LIN {X 0,Y 573.939,Z 295.271,A -85,B 0,C 180,E1 -2262.554,E2 -2262.554} C_VEL
LIN {X 0,Y 573.907,Z 198.013,A -85,B 0,C 180,E1 -2263.779,E2 -2263.779} C_VEL
LIN {X 0,Y 573.417,Z 194.435,A -85,B 0,C 180,E1 -2263.851,E2 -2263.851} C_VEL
LIN {X 0,Y 573.583,Z 173.354,A -85,B 0,C 180,E1 -2266.732,E2 -2266.732} C_VEL
LIN {X 0,Y 573.724,Z 153.908,A -85,B 0,C 180,E1 -2269.398,E2 -2269.398} C_VEL
LIN {X 0,Y 573.977,Z 134.142,A -85,B 0,C 180,E1 -2272.118,E2 -2272.118} C_VEL
LIN {X 0,Y 573.891,Z 125.743,A -85,B 0,C 180,E1 -2273.296,E2 -2273.296} C_VEL
LIN {X 0,Y 573.251,Z 122.082,A -85,B 0,C 180,E1 -2273.865,E2 -2273.865} C_VEL
LIN {X 0,Y 573.218,Z 122.082,A -85,B 0,C 180,E1 -2276.488,E2 -2276.488} C_VEL
LIN {X 0,Y 573.233,Z 122.079,A -85,B 0,C 180,E1 -2278.565,E2 -2278.565} C_VEL
LIN {X 0,Y 573.222,Z 122.078,A -85,B 0,C 180,E1 -2280.994,E2 -2280.994} C_VEL
LIN {X 0,Y 573.266,Z 122.077,A -85,B 0,C 180,E1 -2283.524,E2 -2283.524} C_VEL
LIN {X 0,Y 573.195,Z 122.085,A -85,B 0,C 180,E1 -2286.053,E2 -2286.053} C_VEL
LIN {X 0,Y 573.244,Z 122.074,A -85,B 0,C 180,E1 -2288.702,E2 -2288.702} C_VEL
LIN {X 0,Y 573.225,Z 122.086,A -85,B 0,C 180,E1 -2291.592,E2 -2291.592} C_VEL
LIN {X 0,Y 573.223,Z 122.077,A -85,B 0,C 180,E1 -2294.335,E2 -2294.335} C_VEL
LIN {X 0,Y 573.237,Z 122.084,A -85,B 0,C 180,E1 -2297.359,E2 -2297.359} C_VEL
LIN {X 0,Y 573.233,Z 122.076,A -85,B 0,C 180,E1 -2300.392,E2 -2300.392} C_VEL
LIN {X 0,Y 573.25,Z 122.082,A -85,B 0,C 180,E1 -2303.077,E2 -2303.077} C_VEL
LIN {X 0,Y 573.25,Z 122.075,A -85,B 0,C 180,E1 -2305.67,E2 -2305.67} C_VEL
LIN {X 0,Y 573.224,Z 122.077,A -85,B 0,C 180,E1 -2308.183,E2 -2308.183} C_VEL
LIN {X 0,Y 573.231,Z 122.081,A -85,B 0,C 180,E1 -2310.632,E2 -2310.632} C_VEL
LIN {X 0,Y 573.211,Z 122.079,A -85,B 0,C 180,E1 -2313.513,E2 -2313.513} C_VEL
LIN {X 0,Y 573.192,Z 122.082,A -85,B 0,C 180,E1 -2316.133,E2 -2316.133} C_VEL
LIN {X 0,Y 573.224,Z 122.078,A -85,B 0,C 180,E1 -2319.173,E2 -2319.173} C_VEL
LIN {X 0,Y 573.189,Z 122.08,A -85,B 0,C 180,E1 -2321.41,E2 -2321.41} C_VEL
LIN {X 0,Y 573.199,Z 122.088,A -85,B 0,C 180,E1 -2324.351,E2 -2324.351} C_VEL
LIN {X 0,Y 573.188,Z 122.088,A -85,B 0,C 180,E1 -2326.528,E2 -2326.528} C_VEL
LIN {X 0,Y 573.233,Z 122.075,A -85,B 0,C 180,E1 -2329.403,E2 -2329.403} C_VEL
LIN {X 0,Y 573.209,Z 122.087,A -85,B 0,C 180,E1 -2332.249,E2 -2332.249} C_VEL
LIN {X 0,Y 573.266,Z 122.071,A -85,B 0,C 180,E1 -2335.077,E2 -2335.077} C_VEL
LIN {X 0,Y 573.306,Z 122.073,A -85,B 0,C 180,E1 -2337.892,E2 -2337.892} C_VEL
LIN {X 0,Y 573.314,Z 122.073,A -85,B 0,C 180,E1 -2340,E2 -2340} C_VEL
LIN {X 0,Y 573.268,Z 122.069,A -85,B 0,C 180,E1 -2342.811,E2 -2342.811} C_VEL
LIN {X 0,Y 573.27,Z 122.079,A -85,B 0,C 180,E1 -2345.628,E2 -2345.628} C_VEL
LIN {X 0,Y 573.241,Z 122.073,A -85,B 0,C 180,E1 -2348.46,E2 -2348.46} C_VEL
LIN {X 0,Y 573.271,Z 122.077,A -85,B 0,C 180,E1 -2351.312,E2 -2351.312} C_VEL
LIN {X 0,Y 573.253,Z 122.071,A -85,B 0,C 180,E1 -2354.413,E2 -2354.413} C_VEL
LIN {X 0,Y 573.245,Z 122.08,A -85,B 0,C 180,E1 -2357.112,E2 -2357.112} C_VEL
LIN {X 0,Y 573.232,Z 122.075,A -85,B 0,C 180,E1 -2360.078,E2 -2360.078} C_VEL
LIN {X 0,Y 573.22,Z 122.077,A -85,B 0,C 180,E1 -2362.339,E2 -2362.339} C_VEL
LIN {X 0,Y 573.198,Z 122.079,A -85,B 0,C 180,E1 -2364.344,E2 -2364.344} C_VEL
LIN {X 0,Y 572.559,Z 122.166,A -85,B 0,C 180,E1 -2364.931,E2 -2364.931} C_VEL
LIN {X 0,Y 569.731,Z 122.52,A -85,B 0,C 180,E1 -2365.883,E2 -2365.883} C_VEL
LIN {X 0,Y 567.32,Z 122.82,A -85,B 0,C 180,E1 -2366.648,E2 -2366.648} C_VEL
LIN {X 0,Y 566.274,Z 122.948,A -85,B 0,C 180,E1 -2367.239,E2 -2367.239} C_VEL
LIN {X 0,Y 566.184,Z 122.956,A -85,B 0,C 180,E1 -2367.44,E2 -2367.44} C_VEL
LIN {X 0,Y 566.172,Z 122.955,A -85,B 0,C 180,E1 -2369.771,E2 -2369.771} C_VEL
LIN {X 0,Y 566.201,Z 122.955,A -85,B 0,C 180,E1 -2372.43,E2 -2372.43} C_VEL
LIN {X 0,Y 566.18,Z 122.959,A -85,B 0,C 180,E1 -2374.989,E2 -2374.989} C_VEL
LIN {X 0,Y 566.197,Z 122.952,A -85,B 0,C 180,E1 -2377.461,E2 -2377.461} C_VEL
LIN {X 0,Y 566.208,Z 122.954,A -85,B 0,C 180,E1 -2380.199,E2 -2380.199} C_VEL
LIN {X 0,Y 566.2,Z 122.953,A -85,B 0,C 180,E1 -2383.055,E2 -2383.055} C_VEL
LIN {X 0,Y 566.196,Z 122.957,A -85,B 0,C 180,E1 -2386.049,E2 -2386.049} C_VEL
LIN {X 0,Y 566.206,Z 122.951,A -85,B 0,C 180,E1 -2389.215,E2 -2389.215} C_VEL
LIN {X 0,Y 566.189,Z 122.956,A -85,B 0,C 180,E1 -2391.637,E2 -2391.637} C_VEL
LIN {X 0,Y 566.165,Z 122.962,A -85,B 0,C 180,E1 -2394.308,E2 -2394.308} C_VEL
LIN {X 0,Y 566.224,Z 122.949,A -85,B 0,C 180,E1 -2396.898,E2 -2396.898} C_VEL
LIN {X 0,Y 566.184,Z 122.957,A -85,B 0,C 180,E1 -2399.407,E2 -2399.407} C_VEL
LIN {X 0,Y 566.198,Z 122.961,A -85,B 0,C 180,E1 -2401.856,E2 -2401.856} C_VEL
LIN {X 0,Y 566.217,Z 122.953,A -85,B 0,C 180,E1 -2404.251,E2 -2404.251} C_VEL
LIN {X 0,Y 566.24,Z 123.02,A -85,B 0,C 180,E1 -2406.598,E2 -2406.598} C_VEL
LIN {X 0,Y 566.394,Z 130.26,A -85,B 0,C 180,E1 -2407.954,E2 -2407.954} C_VEL
LIN {X 0,Y 566.229,Z 145.729,A -85,B 0,C 180,E1 -2410.874,E2 -2410.874} C_VEL
LIN {X 0,Y 566.186,Z 146.658,A -85,B 0,C 180,E1 -2411.05,E2 -2411.05} C_VEL
LIN {X 0,Y 567.206,Z 153.44,A -85,B 0,C 180,E1 -2411.169,E2 -2411.169} C_VEL
LIN {X 0,Y 566.897,Z 253.478,A -85,B 0,C 180,E1 -2412.457,E2 -2412.457} C_VEL
LIN {X 0,Y 566.788,Z 267.319,A -85,B 0,C 180,E1 -2412.796,E2 -2412.796} C_VEL
LIN {X 0,Y 566.722,Z 279.942,A -85,B 0,C 180,E1 -2413.258,E2 -2413.258} C_VEL
LIN {X 0,Y 566.568,Z 292.491,A -85,B 0,C 180,E1 -2413.885,E2 -2413.885} C_VEL
LIN {X 0,Y 566.436,Z 303.91,A -85,B 0,C 180,E1 -2414.62,E2 -2414.62} C_VEL
LIN {X 0,Y 566.278,Z 314.5,A -85,B 0,C 180,E1 -2415.479,E2 -2415.479} C_VEL
LIN {X 0,Y 566.22,Z 323.325,A -85,B 0,C 180,E1 -2416.359,E2 -2416.359} C_VEL
LIN {X 0,Y 566.067,Z 332.259,A -85,B 0,C 180,E1 -2417.451,E2 -2417.451} C_VEL
LIN {X 0,Y 566.016,Z 339.371,A -85,B 0,C 180,E1 -2418.541,E2 -2418.541} C_VEL
LIN {X 0,Y 565.933,Z 345.026,A -85,B 0,C 180,E1 -2419.626,E2 -2419.626} C_VEL
LIN {X 0,Y 565.88,Z 349.456,A -85,B 0,C 180,E1 -2420.708,E2 -2420.708} C_VEL
LIN {X 0,Y 565.891,Z 351.793,A -85,B 0,C 180,E1 -2421.429,E2 -2421.429} C_VEL
LIN {X 0,Y 565.891,Z 353.691,A -85,B 0,C 180,E1 -2422.148,E2 -2422.148} C_VEL
LIN {X 0,Y 565.923,Z 356.006,A -85,B 0,C 180,E1 -2423.463,E2 -2423.463} C_VEL
LIN {X 0,Y 565.899,Z 356.763,A -85,B 0,C 180,E1 -2424.297,E2 -2424.297} C_VEL
LIN {X 0,Y 565.849,Z 356.998,A -85,B 0,C 180,E1 -2425.012,E2 -2425.012} C_VEL
LIN {X 0,Y 565.912,Z 356.806,A -85,B 0,C 180,E1 -2425.726,E2 -2425.726} C_VEL
LIN {X 0,Y 565.911,Z 356.216,A -85,B 0,C 180,E1 -2426.439,E2 -2426.439} C_VEL
LIN {X 0,Y 565.841,Z 353.871,A -85,B 0,C 180,E1 -2427.864,E2 -2427.864} C_VEL
LIN {X 0,Y 565.888,Z 350.984,A -85,B 0,C 180,E1 -2428.932,E2 -2428.932} C_VEL
LIN {X 0,Y 565.905,Z 347.081,A -85,B 0,C 180,E1 -2429.999,E2 -2429.999} C_VEL
LIN {X 0,Y 565.991,Z 342.057,A -85,B 0,C 180,E1 -2431.067,E2 -2431.067} C_VEL
LIN {X 0,Y 565.977,Z 335.764,A -85,B 0,C 180,E1 -2432.134,E2 -2432.134} C_VEL
LIN {X 0,Y 566.169,Z 327.896,A -85,B 0,C 180,E1 -2433.201,E2 -2433.201} C_VEL
LIN {X 0,Y 566.237,Z 319.912,A -85,B 0,C 180,E1 -2434.092,E2 -2434.092} C_VEL
LIN {X 0,Y 566.321,Z 310.198,A -85,B 0,C 180,E1 -2434.983,E2 -2434.983} C_VEL
LIN {X 0,Y 566.461,Z 299.366,A -85,B 0,C 180,E1 -2435.785,E2 -2435.785} C_VEL
LIN {X 0,Y 566.658,Z 287.581,A -85,B 0,C 180,E1 -2436.47,E2 -2436.47} C_VEL
LIN {X 0,Y 566.766,Z 275.517,A -85,B 0,C 180,E1 -2437.011,E2 -2437.011} C_VEL
LIN {X 0,Y 566.847,Z 263.545,A -85,B 0,C 180,E1 -2437.405,E2 -2437.405} C_VEL
LIN {X 0,Y 566.903,Z 250.677,A -85,B 0,C 180,E1 -2437.68,E2 -2437.68} C_VEL
LIN {X 0,Y 567.048,Z 151.584,A -85,B 0,C 180,E1 -2438.949,E2 -2438.949} C_VEL
LIN {X 0,Y 566.192,Z 146.551,A -85,B 0,C 180,E1 -2439.06,E2 -2439.06} C_VEL
LIN {X 0,Y 566.372,Z 131.992,A -85,B 0,C 180,E1 -2441.814,E2 -2441.814} C_VEL
LIN {X 0,Y 566.232,Z 122.953,A -85,B 0,C 180,E1 -2443.525,E2 -2443.525} C_VEL
LIN {X 0,Y 566.213,Z 122.957,A -85,B 0,C 180,E1 -2446.587,E2 -2446.587} C_VEL
LIN {X 0,Y 566.203,Z 122.952,A -85,B 0,C 180,E1 -2449.58,E2 -2449.58} C_VEL
LIN {X 0,Y 566.194,Z 122.957,A -85,B 0,C 180,E1 -2451.861,E2 -2451.861} C_VEL
LIN {X 0,Y 566.218,Z 122.949,A -85,B 0,C 180,E1 -2455.029,E2 -2455.029} C_VEL
LIN {X 0,Y 566.192,Z 122.954,A -85,B 0,C 180,E1 -2457.339,E2 -2457.339} C_VEL
LIN {X 0,Y 566.198,Z 122.959,A -85,B 0,C 180,E1 -2459.768,E2 -2459.768} C_VEL
LIN {X 0,Y 566.2,Z 122.954,A -85,B 0,C 180,E1 -2462.429,E2 -2462.429} C_VEL
LIN {X 0,Y 566.176,Z 122.955,A -85,B 0,C 180,E1 -2464.988,E2 -2464.988} C_VEL
LIN {X 0,Y 566.192,Z 122.959,A -85,B 0,C 180,E1 -2467.46,E2 -2467.46} C_VEL
LIN {X 0,Y 566.204,Z 122.953,A -85,B 0,C 180,E1 -2470.198,E2 -2470.198} C_VEL
LIN {X 0,Y 566.194,Z 122.956,A -85,B 0,C 180,E1 -2473.053,E2 -2473.053} C_VEL
LIN {X 0,Y 566.187,Z 122.955,A -85,B 0,C 180,E1 -2476.048,E2 -2476.048} C_VEL
LIN {X 0,Y 566.196,Z 122.96,A -85,B 0,C 180,E1 -2479.214,E2 -2479.214} C_VEL
LIN {X 0,Y 566.173,Z 122.959,A -85,B 0,C 180,E1 -2481.635,E2 -2481.635} C_VEL
LIN {X 0,Y 566.153,Z 122.958,A -85,B 0,C 180,E1 -2484.307,E2 -2484.307} C_VEL
LIN {X 0,Y 566.189,Z 122.961,A -85,B 0,C 180,E1 -2486.896,E2 -2486.896} C_VEL
LIN {X 0,Y 566.161,Z 122.96,A -85,B 0,C 180,E1 -2489.406,E2 -2489.406} C_VEL
LIN {X 0,Y 566.183,Z 122.954,A -85,B 0,C 180,E1 -2491.856,E2 -2491.856} C_VEL
LIN {X 0,Y 566.181,Z 122.956,A -85,B 0,C 180,E1 -2494.249,E2 -2494.249} C_VEL
LIN {X 0,Y 566.151,Z 122.96,A -85,B 0,C 180,E1 -2497.367,E2 -2497.367} C_VEL
LIN {X 0,Y 566.188,Z 122.954,A -85,B 0,C 180,E1 -2499.662,E2 -2499.662} C_VEL
LIN {X 0,Y 566.161,Z 122.958,A -85,B 0,C 180,E1 -2501.92,E2 -2501.92} C_VEL
LIN {X 0,Y 566.169,Z 122.96,A -85,B 0,C 180,E1 -2504.89,E2 -2504.89} C_VEL
LIN {X 0,Y 566.168,Z 122.958,A -85,B 0,C 180,E1 -2507.817,E2 -2507.817} C_VEL
LIN {X 0,Y 566.157,Z 122.962,A -85,B 0,C 180,E1 -2509.992,E2 -2509.992} C_VEL
LIN {X 0,Y 566.196,Z 122.954,A -85,B 0,C 180,E1 -2512.87,E2 -2512.87} C_VEL
LIN {X 0,Y 566.24,Z 122.948,A -85,B 0,C 180,E1 -2515.016,E2 -2515.016} C_VEL
LIN {X 0,Y 566.269,Z 122.95,A -85,B 0,C 180,E1 -2517.866,E2 -2517.866} C_VEL
LIN {X 0,Y 566.273,Z 122.951,A -85,B 0,C 180,E1 -2520,E2 -2520} C_VEL
LIN {X 0,Y 566.228,Z 122.949,A -85,B 0,C 180,E1 -2522.846,E2 -2522.846} C_VEL
LIN {X 0,Y 566.237,Z 122.956,A -85,B 0,C 180,E1 -2525.698,E2 -2525.698} C_VEL
LIN {X 0,Y 566.184,Z 122.955,A -85,B 0,C 180,E1 -2528.566,E2 -2528.566} C_VEL
LIN {X 0,Y 566.226,Z 122.956,A -85,B 0,C 180,E1 -2531.455,E2 -2531.455} C_VEL
LIN {X 0,Y 566.197,Z 122.953,A -85,B 0,C 180,E1 -2534.497,E2 -2534.497} C_VEL
LIN {X 0,Y 566.174,Z 122.964,A -85,B 0,C 180,E1 -2537.332,E2 -2537.332} C_VEL
LIN {X 0,Y 566.187,Z 122.96,A -85,B 0,C 180,E1 -2539.582,E2 -2539.582} C_VEL
LIN {X 0,Y 566.174,Z 122.957,A -85,B 0,C 180,E1 -2541.863,E2 -2541.863} C_VEL
LIN {X 0,Y 566.166,Z 122.964,A -85,B 0,C 180,E1 -2545.022,E2 -2545.022} C_VEL
LIN {X 0,Y 566.198,Z 122.958,A -85,B 0,C 180,E1 -2547.34,E2 -2547.34} C_VEL
LIN {X 0,Y 566.185,Z 122.955,A -85,B 0,C 180,E1 -2549.77,E2 -2549.77} C_VEL
LIN {X 0,Y 566.192,Z 122.956,A -85,B 0,C 180,E1 -2552.431,E2 -2552.431} C_VEL
LIN {X 0,Y 566.171,Z 122.963,A -85,B 0,C 180,E1 -2554.99,E2 -2554.99} C_VEL
LIN {X 0,Y 566.187,Z 122.955,A -85,B 0,C 180,E1 -2557.462,E2 -2557.462} C_VEL
LIN {X 0,Y 566.198,Z 122.955,A -85,B 0,C 180,E1 -2560.2,E2 -2560.2} C_VEL
LIN {X 0,Y 566.194,Z 122.955,A -85,B 0,C 180,E1 -2563.055,E2 -2563.055} C_VEL
LIN {X 0,Y 566.187,Z 122.957,A -85,B 0,C 180,E1 -2566.05,E2 -2566.05} C_VEL
LIN {X 0,Y 566.198,Z 122.952,A -85,B 0,C 180,E1 -2569.216,E2 -2569.216} C_VEL
LIN {X 0,Y 566.181,Z 122.955,A -85,B 0,C 180,E1 -2571.638,E2 -2571.638} C_VEL
LIN {X 0,Y 566.158,Z 122.965,A -85,B 0,C 180,E1 -2574.309,E2 -2574.309} C_VEL
LIN {X 0,Y 566.216,Z 122.95,A -85,B 0,C 180,E1 -2576.899,E2 -2576.899} C_VEL
LIN {X 0,Y 566.183,Z 122.955,A -85,B 0,C 180,E1 -2579.409,E2 -2579.409} C_VEL
LIN {X 0,Y 566.209,Z 122.959,A -85,B 0,C 180,E1 -2581.858,E2 -2581.858} C_VEL
LIN {X 0,Y 566.212,Z 122.954,A -85,B 0,C 180,E1 -2584.252,E2 -2584.252} C_VEL
LIN {X 0,Y 566.227,Z 122.976,A -85,B 0,C 180,E1 -2586.017,E2 -2586.017} C_VEL
LIN {X 0,Y 567.072,Z 128.443,A -85,B 0,C 180,E1 -2586.829,E2 -2586.829} C_VEL
LIN {X 0,Y 566.876,Z 147.438,A -85,B 0,C 180,E1 -2589.499,E2 -2589.499} C_VEL
LIN {X 0,Y 566.649,Z 167.761,A -85,B 0,C 180,E1 -2592.311,E2 -2592.311} C_VEL
LIN {X 0,Y 566.437,Z 187.958,A -85,B 0,C 180,E1 -2595.081,E2 -2595.081} C_VEL
LIN {X 0,Y 566.423,Z 194.528,A -85,B 0,C 180,E1 -2595.988,E2 -2595.988} C_VEL
LIN {X 0,Y 567.162,Z 201.308,A -85,B 0,C 180,E1 -2596.096,E2 -2596.096} C_VEL
LIN {X 0,Y 566.937,Z 302.989,A -85,B 0,C 180,E1 -2597.403,E2 -2597.403} C_VEL
LIN {X 0,Y 566.838,Z 316.245,A -85,B 0,C 180,E1 -2597.719,E2 -2597.719} C_VEL
LIN {X 0,Y 566.719,Z 328.398,A -85,B 0,C 180,E1 -2598.149,E2 -2598.149} C_VEL
LIN {X 0,Y 566.606,Z 340.204,A -85,B 0,C 180,E1 -2598.711,E2 -2598.711} C_VEL
LIN {X 0,Y 566.439,Z 352.207,A -85,B 0,C 180,E1 -2599.456,E2 -2599.456} C_VEL
LIN {X 0,Y 566.325,Z 362.614,A -85,B 0,C 180,E1 -2600.266,E2 -2600.266} C_VEL
LIN {X 0,Y 566.207,Z 371.121,A -85,B 0,C 180,E1 -2601.075,E2 -2601.075} C_VEL
LIN {X 0,Y 566.112,Z 378.967,A -85,B 0,C 180,E1 -2601.972,E2 -2601.972} C_VEL
LIN {X 0,Y 566.001,Z 386.627,A -85,B 0,C 180,E1 -2603.047,E2 -2603.047} C_VEL
LIN {X 0,Y 566.004,Z 393.683,A -85,B 0,C 180,E1 -2604.3,E2 -2604.3} C_VEL
LIN {X 0,Y 565.933,Z 398.375,A -85,B 0,C 180,E1 -2605.371,E2 -2605.371} C_VEL
LIN {X 0,Y 565.927,Z 401.96,A -85,B 0,C 180,E1 -2606.441,E2 -2606.441} C_VEL
LIN {X 0,Y 565.878,Z 403.809,A -85,B 0,C 180,E1 -2607.153,E2 -2607.153} C_VEL
LIN {X 0,Y 565.846,Z 406.185,A -85,B 0,C 180,E1 -2608.577,E2 -2608.577} C_VEL
LIN {X 0,Y 565.839,Z 407,A -85,B 0,C 180,E1 -2610.001,E2 -2610.001} C_VEL
LIN {X 0,Y 565.846,Z 406.184,A -85,B 0,C 180,E1 -2611.424,E2 -2611.424} C_VEL
LIN {X 0,Y 565.878,Z 403.809,A -85,B 0,C 180,E1 -2612.848,E2 -2612.848} C_VEL
LIN {X 0,Y 565.926,Z 400.894,A -85,B 0,C 180,E1 -2613.917,E2 -2613.917} C_VEL
LIN {X 0,Y 565.878,Z 396.946,A -85,B 0,C 180,E1 -2614.988,E2 -2614.988} C_VEL
LIN {X 0,Y 566.002,Z 391.864,A -85,B 0,C 180,E1 -2616.059,E2 -2616.059} C_VEL
LIN {X 0,Y 566.041,Z 385.463,A -85,B 0,C 180,E1 -2617.133,E2 -2617.133} C_VEL
LIN {X 0,Y 566.134,Z 377.473,A -85,B 0,C 180,E1 -2618.208,E2 -2618.208} C_VEL
LIN {X 0,Y 566.229,Z 369.329,A -85,B 0,C 180,E1 -2619.106,E2 -2619.106} C_VEL
LIN {X 0,Y 566.348,Z 359.392,A -85,B 0,C 180,E1 -2620.005,E2 -2620.005} C_VEL
LIN {X 0,Y 566.536,Z 348.283,A -85,B 0,C 180,E1 -2620.808,E2 -2620.808} C_VEL
LIN {X 0,Y 566.613,Z 337.163,A -85,B 0,C 180,E1 -2621.447,E2 -2621.447} C_VEL
LIN {X 0,Y 566.746,Z 324.966,A -85,B 0,C 180,E1 -2621.989,E2 -2621.989} C_VEL
LIN {X 0,Y 566.888,Z 312.154,A -85,B 0,C 180,E1 -2622.394,E2 -2622.394} C_VEL
LIN {X 0,Y 566.998,Z 300.072,A -85,B 0,C 180,E1 -2622.642,E2 -2622.642} C_VEL
LIN {X 0,Y 567.061,Z 198.889,A -85,B 0,C 180,E1 -2623.938,E2 -2623.938} C_VEL
LIN {X 0,Y 566.421,Z 194.435,A -85,B 0,C 180,E1 -2624.025,E2 -2624.025} C_VEL
LIN {X 0,Y 566.628,Z 171.832,A -85,B 0,C 180,E1 -2627.128,E2 -2627.128} C_VEL
LIN {X 0,Y 566.86,Z 150.118,A -85,B 0,C 180,E1 -2630.124,E2 -2630.124} C_VEL
LIN {X 0,Y 567.045,Z 129.747,A -85,B 0,C 180,E1 -2632.981,E2 -2632.981} C_VEL
LIN {X 0,Y 566.465,Z 124.281,A -85,B 0,C 180,E1 -2633.78,E2 -2633.78} C_VEL
LIN {X 0,Y 566.212,Z 122.959,A -85,B 0,C 180,E1 -2633.985,E2 -2633.985} C_VEL
LIN {X 0,Y 566.188,Z 122.956,A -85,B 0,C 180,E1 -2636.655,E2 -2636.655} C_VEL
LIN {X 0,Y 566.181,Z 122.956,A -85,B 0,C 180,E1 -2638.954,E2 -2638.954} C_VEL
LIN {X 0,Y 566.192,Z 122.957,A -85,B 0,C 180,E1 -2641.422,E2 -2641.422} C_VEL
LIN {X 0,Y 566.211,Z 122.958,A -85,B 0,C 180,E1 -2643.956,E2 -2643.956} C_VEL
LIN {X 0,Y 566.184,Z 122.953,A -85,B 0,C 180,E1 -2646.571,E2 -2646.571} C_VEL
LIN {X 0,Y 566.219,Z 122.958,A -85,B 0,C 180,E1 -2649.686,E2 -2649.686} C_VEL
LIN {X 0,Y 566.193,Z 122.954,A -85,B 0,C 180,E1 -2652.916,E2 -2652.916} C_VEL
LIN {X 0,Y 566.16,Z 122.959,A -85,B 0,C 180,E1 -2655.96,E2 -2655.96} C_VEL
LIN {X 0,Y 566.179,Z 122.955,A -85,B 0,C 180,E1 -2658.14,E2 -2658.14} C_VEL
LIN {X 0,Y 566.209,Z 122.953,A -85,B 0,C 180,E1 -2660.726,E2 -2660.726} C_VEL
LIN {X 0,Y 566.191,Z 122.958,A -85,B 0,C 180,E1 -2663.429,E2 -2663.429} C_VEL
LIN {X 0,Y 566.196,Z 122.953,A -85,B 0,C 180,E1 -2666.268,E2 -2666.268} C_VEL
LIN {X 0,Y 566.18,Z 122.963,A -85,B 0,C 180,E1 -2668.925,E2 -2668.925} C_VEL
LIN {X 0,Y 566.148,Z 122.958,A -85,B 0,C 180,E1 -2671.854,E2 -2671.854} C_VEL
LIN {X 0,Y 566.187,Z 122.955,A -85,B 0,C 180,E1 -2674.25,E2 -2674.25} C_VEL
LIN {X 0,Y 566.144,Z 122.959,A -85,B 0,C 180,E1 -2677.367,E2 -2677.367} C_VEL
LIN {X 0,Y 566.167,Z 122.955,A -85,B 0,C 180,E1 -2679.661,E2 -2679.661} C_VEL
LIN {X 0,Y 566.16,Z 122.957,A -85,B 0,C 180,E1 -2681.92,E2 -2681.92} C_VEL
LIN {X 0,Y 566.176,Z 122.956,A -85,B 0,C 180,E1 -2684.89,E2 -2684.89} C_VEL
LIN {X 0,Y 566.16,Z 122.958,A -85,B 0,C 180,E1 -2687.817,E2 -2687.817} C_VEL
LIN {X 0,Y 566.151,Z 122.963,A -85,B 0,C 180,E1 -2689.992,E2 -2689.992} C_VEL
LIN {X 0,Y 566.179,Z 122.955,A -85,B 0,C 180,E1 -2692.87,E2 -2692.87} C_VEL
LIN {X 0,Y 566.242,Z 122.946,A -85,B 0,C 180,E1 -2695.016,E2 -2695.016} C_VEL
LIN {X 0,Y 566.276,Z 122.948,A -85,B 0,C 180,E1 -2697.866,E2 -2697.866} C_VEL
LIN {X 0,Y 566.283,Z 122.949,A -85,B 0,C 180,E1 -2700,E2 -2700} C_VEL
LIN {X 0,Y 566.237,Z 122.945,A -85,B 0,C 180,E1 -2702.846,E2 -2702.846} C_VEL
LIN {X 0,Y 566.237,Z 122.956,A -85,B 0,C 180,E1 -2705.699,E2 -2705.699} C_VEL
LIN {X 0,Y 566.193,Z 122.95,A -85,B 0,C 180,E1 -2708.566,E2 -2708.566} C_VEL
LIN {X 0,Y 566.238,Z 122.956,A -85,B 0,C 180,E1 -2711.455,E2 -2711.455} C_VEL
LIN {X 0,Y 566.209,Z 122.949,A -85,B 0,C 180,E1 -2714.497,E2 -2714.497} C_VEL
LIN {X 0,Y 566.186,Z 122.962,A -85,B 0,C 180,E1 -2717.332,E2 -2717.332} C_VEL
LIN {X 0,Y 566.198,Z 122.955,A -85,B 0,C 180,E1 -2719.581,E2 -2719.581} C_VEL
LIN {X 0,Y 566.185,Z 122.954,A -85,B 0,C 180,E1 -2721.863,E2 -2721.863} C_VEL
LIN {X 0,Y 566.178,Z 122.962,A -85,B 0,C 180,E1 -2725.021,E2 -2725.021} C_VEL
LIN {X 0,Y 566.184,Z 122.956,A -85,B 0,C 180,E1 -2727.44,E2 -2727.44} C_VEL
LIN {X 0,Y 565.502,Z 123.04,A -85,B 0,C 180,E1 -2728.033,E2 -2728.033} C_VEL
LIN {X 0,Y 562.638,Z 123.403,A -85,B 0,C 180,E1 -2728.997,E2 -2728.997} C_VEL
LIN {X 0,Y 560.232,Z 123.699,A -85,B 0,C 180,E1 -2729.773,E2 -2729.773} C_VEL
LIN {X 0,Y 559.208,Z 123.825,A -85,B 0,C 180,E1 -2730.372,E2 -2730.372} C_VEL
LIN {X 0,Y 559.129,Z 123.834,A -85,B 0,C 180,E1 -2730.574,E2 -2730.574} C_VEL
LIN {X 0,Y 559.152,Z 123.838,A -85,B 0,C 180,E1 -2732.716,E2 -2732.716} C_VEL
LIN {X 0,Y 559.128,Z 123.833,A -85,B 0,C 180,E1 -2735.324,E2 -2735.324} C_VEL
LIN {X 0,Y 559.132,Z 123.834,A -85,B 0,C 180,E1 -2738.018,E2 -2738.018} C_VEL
LIN {X 0,Y 559.157,Z 123.831,A -85,B 0,C 180,E1 -2740.813,E2 -2740.813} C_VEL
LIN {X 0,Y 559.14,Z 123.832,A -85,B 0,C 180,E1 -2743.734,E2 -2743.734} C_VEL
LIN {X 0,Y 559.145,Z 123.833,A -85,B 0,C 180,E1 -2746.804,E2 -2746.804} C_VEL
LIN {X 0,Y 559.158,Z 123.829,A -85,B 0,C 180,E1 -2749.188,E2 -2749.188} C_VEL
LIN {X 0,Y 559.136,Z 123.839,A -85,B 0,C 180,E1 -2751.982,E2 -2751.982} C_VEL
LIN {X 0,Y 559.134,Z 123.833,A -85,B 0,C 180,E1 -2754.787,E2 -2754.787} C_VEL
LIN {X 0,Y 559.159,Z 123.831,A -85,B 0,C 180,E1 -2757.365,E2 -2757.365} C_VEL
LIN {X 0,Y 559.152,Z 123.835,A -85,B 0,C 180,E1 -2760.143,E2 -2760.143} C_VEL
LIN {X 0,Y 559.171,Z 123.831,A -85,B 0,C 180,E1 -2763.173,E2 -2763.173} C_VEL
LIN {X 0,Y 559.165,Z 123.837,A -85,B 0,C 180,E1 -2765.495,E2 -2765.495} C_VEL
LIN {X 0,Y 559.231,Z 124.03,A -85,B 0,C 180,E1 -2766.551,E2 -2766.551} C_VEL
LIN {X 0,Y 559.381,Z 132.609,A -85,B 0,C 180,E1 -2768.174,E2 -2768.174} C_VEL
LIN {X 0,Y 559.224,Z 146.903,A -85,B 0,C 180,E1 -2770.868,E2 -2770.868} C_VEL
LIN {X 0,Y 560.315,Z 154.161,A -85,B 0,C 180,E1 -2771.001,E2 -2771.001} C_VEL
LIN {X 0,Y 559.987,Z 253.898,A -85,B 0,C 180,E1 -2772.304,E2 -2772.304} C_VEL
LIN {X 0,Y 559.868,Z 267.225,A -85,B 0,C 180,E1 -2772.635,E2 -2772.635} C_VEL
LIN {X 0,Y 559.779,Z 278.994,A -85,B 0,C 180,E1 -2773.064,E2 -2773.064} C_VEL
LIN {X 0,Y 559.626,Z 291.434,A -85,B 0,C 180,E1 -2773.68,E2 -2773.68} C_VEL
LIN {X 0,Y 559.441,Z 303.006,A -85,B 0,C 180,E1 -2774.423,E2 -2774.423} C_VEL
LIN {X 0,Y 559.27,Z 313.628,A -85,B 0,C 180,E1 -2775.276,E2 -2775.276} C_VEL
LIN {X 0,Y 559.17,Z 322.745,A -85,B 0,C 180,E1 -2776.184,E2 -2776.184} C_VEL
LIN {X 0,Y 559.002,Z 331.777,A -85,B 0,C 180,E1 -2777.289,E2 -2777.289} C_VEL
LIN {X 0,Y 558.962,Z 339.011,A -85,B 0,C 180,E1 -2778.394,E2 -2778.394} C_VEL
LIN {X 0,Y 558.86,Z 344.741,A -85,B 0,C 180,E1 -2779.493,E2 -2779.493} C_VEL
LIN {X 0,Y 558.797,Z 349.237,A -85,B 0,C 180,E1 -2780.589,E2 -2780.589} C_VEL
LIN {X 0,Y 558.808,Z 351.605,A -85,B 0,C 180,E1 -2781.319,E2 -2781.319} C_VEL
LIN {X 0,Y 558.811,Z 353.536,A -85,B 0,C 180,E1 -2782.047,E2 -2782.047} C_VEL
LIN {X 0,Y 558.799,Z 355.027,A -85,B 0,C 180,E1 -2782.774,E2 -2782.774} C_VEL
LIN {X 0,Y 558.847,Z 356.069,A -85,B 0,C 180,E1 -2783.501,E2 -2783.501} C_VEL
LIN {X 0,Y 558.763,Z 356.985,A -85,B 0,C 180,E1 -2784.948,E2 -2784.948} C_VEL
LIN {X 0,Y 558.805,Z 356.847,A -85,B 0,C 180,E1 -2785.672,E2 -2785.672} C_VEL
LIN {X 0,Y 558.82,Z 356.285,A -85,B 0,C 180,E1 -2786.394,E2 -2786.394} C_VEL
LIN {X 0,Y 558.795,Z 355.337,A -85,B 0,C 180,E1 -2787.116,E2 -2787.116} C_VEL
LIN {X 0,Y 558.747,Z 353.998,A -85,B 0,C 180,E1 -2787.837,E2 -2787.837} C_VEL
LIN {X 0,Y 558.796,Z 351.169,A -85,B 0,C 180,E1 -2788.918,E2 -2788.918} C_VEL
LIN {X 0,Y 558.81,Z 347.329,A -85,B 0,C 180,E1 -2789.999,E2 -2789.999} C_VEL
LIN {X 0,Y 558.916,Z 342.372,A -85,B 0,C 180,E1 -2791.08,E2 -2791.08} C_VEL
LIN {X 0,Y 558.894,Z 336.167,A -85,B 0,C 180,E1 -2792.161,E2 -2792.161} C_VEL
LIN {X 0,Y 559.119,Z 328.411,A -85,B 0,C 180,E1 -2793.242,E2 -2793.242} C_VEL
LIN {X 0,Y 559.2,Z 320.529,A -85,B 0,C 180,E1 -2794.143,E2 -2794.143} C_VEL
LIN {X 0,Y 559.305,Z 310.937,A -85,B 0,C 180,E1 -2795.045,E2 -2795.045} C_VEL
LIN {X 0,Y 559.445,Z 300.33,A -85,B 0,C 180,E1 -2795.858,E2 -2795.858} C_VEL
LIN {X 0,Y 559.674,Z 288.785,A -85,B 0,C 180,E1 -2796.556,E2 -2796.556} C_VEL
LIN {X 0,Y 559.823,Z 276.55,A -85,B 0,C 180,E1 -2797.125,E2 -2797.125} C_VEL
LIN {X 0,Y 559.909,Z 264.089,A -85,B 0,C 180,E1 -2797.55,E2 -2797.55} C_VEL
LIN {X 0,Y 559.99,Z 252.007,A -85,B 0,C 180,E1 -2797.821,E2 -2797.821} C_VEL
LIN {X 0,Y 560.197,Z 152.604,A -85,B 0,C 180,E1 -2799.113,E2 -2799.113} C_VEL
LIN {X 0,Y 559.216,Z 146.913,A -85,B 0,C 180,E1 -2799.22,E2 -2799.22} C_VEL
LIN {X 0,Y 559.362,Z 132.406,A -85,B 0,C 180,E1 -2801.964,E2 -2801.964} C_VEL
LIN {X 0,Y 559.195,Z 123.845,A -85,B 0,C 180,E1 -2803.583,E2 -2803.583} C_VEL
LIN {X 0,Y 559.164,Z 123.834,A -85,B 0,C 180,E1 -2806.051,E2 -2806.051} C_VEL
LIN {X 0,Y 559.162,Z 123.829,A -85,B 0,C 180,E1 -2809.073,E2 -2809.073} C_VEL
LIN {X 0,Y 559.157,Z 123.83,A -85,B 0,C 180,E1 -2811.549,E2 -2811.549} C_VEL
LIN {X 0,Y 559.156,Z 123.833,A -85,B 0,C 180,E1 -2814.504,E2 -2814.504} C_VEL
LIN {X 0,Y 559.163,Z 123.829,A -85,B 0,C 180,E1 -2816.902,E2 -2816.902} C_VEL
LIN {X 0,Y 559.146,Z 123.838,A -85,B 0,C 180,E1 -2819.856,E2 -2819.856} C_VEL
LIN {X 0,Y 559.154,Z 123.83,A -85,B 0,C 180,E1 -2822.714,E2 -2822.714} C_VEL
LIN {X 0,Y 559.124,Z 123.837,A -85,B 0,C 180,E1 -2825.323,E2 -2825.323} C_VEL
LIN {X 0,Y 559.128,Z 123.837,A -85,B 0,C 180,E1 -2828.016,E2 -2828.016} C_VEL
LIN {X 0,Y 559.15,Z 123.831,A -85,B 0,C 180,E1 -2830.811,E2 -2830.811} C_VEL
LIN {X 0,Y 559.132,Z 123.838,A -85,B 0,C 180,E1 -2833.733,E2 -2833.733} C_VEL
LIN {X 0,Y 559.136,Z 123.834,A -85,B 0,C 180,E1 -2836.803,E2 -2836.803} C_VEL
LIN {X 0,Y 559.147,Z 123.838,A -85,B 0,C 180,E1 -2839.186,E2 -2839.186} C_VEL
LIN {X 0,Y 559.122,Z 123.835,A -85,B 0,C 180,E1 -2841.981,E2 -2841.981} C_VEL
LIN {X 0,Y 559.122,Z 123.838,A -85,B 0,C 180,E1 -2844.786,E2 -2844.786} C_VEL
LIN {X 0,Y 559.142,Z 123.836,A -85,B 0,C 180,E1 -2847.364,E2 -2847.364} C_VEL
LIN {X 0,Y 559.132,Z 123.833,A -85,B 0,C 180,E1 -2850.143,E2 -2850.143} C_VEL
LIN {X 0,Y 559.15,Z 123.835,A -85,B 0,C 180,E1 -2853.174,E2 -2853.174} C_VEL
LIN {X 0,Y 559.104,Z 123.837,A -85,B 0,C 180,E1 -2855.492,E2 -2855.492} C_VEL
LIN {X 0,Y 559.159,Z 123.837,A -85,B 0,C 180,E1 -2858.623,E2 -2858.623} C_VEL
LIN {X 0,Y 559.143,Z 123.836,A -85,B 0,C 180,E1 -2860.925,E2 -2860.925} C_VEL
LIN {X 0,Y 559.122,Z 123.836,A -85,B 0,C 180,E1 -2863.946,E2 -2863.946} C_VEL
LIN {X 0,Y 559.131,Z 123.839,A -85,B 0,C 180,E1 -2866.183,E2 -2866.183} C_VEL
LIN {X 0,Y 559.177,Z 123.828,A -85,B 0,C 180,E1 -2869.133,E2 -2869.133} C_VEL
LIN {X 0,Y 559.173,Z 123.834,A -85,B 0,C 180,E1 -2872.053,E2 -2872.053} C_VEL
LIN {X 0,Y 559.217,Z 123.823,A -85,B 0,C 180,E1 -2874.953,E2 -2874.953} C_VEL
LIN {X 0,Y 559.239,Z 123.826,A -85,B 0,C 180,E1 -2877.839,E2 -2877.839} C_VEL
LIN {X 0,Y 559.242,Z 123.827,A -85,B 0,C 180,E1 -2880,E2 -2880} C_VEL
LIN {X 0,Y 559.196,Z 123.825,A -85,B 0,C 180,E1 -2882.882,E2 -2882.882} C_VEL
LIN {X 0,Y 559.205,Z 123.831,A -85,B 0,C 180,E1 -2885.77,E2 -2885.77} C_VEL
LIN {X 0,Y 559.148,Z 123.831,A -85,B 0,C 180,E1 -2888.675,E2 -2888.675} C_VEL
LIN {X 0,Y 559.187,Z 123.833,A -85,B 0,C 180,E1 -2891.601,E2 -2891.601} C_VEL
LIN {X 0,Y 559.145,Z 123.831,A -85,B 0,C 180,E1 -2894.579,E2 -2894.579} C_VEL
LIN {X 0,Y 559.118,Z 123.841,A -85,B 0,C 180,E1 -2897.558,E2 -2897.558} C_VEL
LIN {X 0,Y 559.15,Z 123.833,A -85,B 0,C 180,E1 -2899.838,E2 -2899.838} C_VEL
LIN {X 0,Y 559.122,Z 123.834,A -85,B 0,C 180,E1 -2902.154,E2 -2902.154} C_VEL
LIN {X 0,Y 559.127,Z 123.841,A -85,B 0,C 180,E1 -2905.179,E2 -2905.179} C_VEL
LIN {X 0,Y 559.137,Z 123.833,A -85,B 0,C 180,E1 -2907.715,E2 -2907.715} C_VEL
LIN {X 0,Y 559.139,Z 123.832,A -85,B 0,C 180,E1 -2910.184,E2 -2910.184} C_VEL
LIN {X 0,Y 559.141,Z 123.838,A -85,B 0,C 180,E1 -2912.716,E2 -2912.716} C_VEL
LIN {X 0,Y 559.118,Z 123.837,A -85,B 0,C 180,E1 -2915.325,E2 -2915.325} C_VEL
LIN {X 0,Y 559.123,Z 123.834,A -85,B 0,C 180,E1 -2918.019,E2 -2918.019} C_VEL
LIN {X 0,Y 559.147,Z 123.837,A -85,B 0,C 180,E1 -2920.813,E2 -2920.813} C_VEL
LIN {X 0,Y 559.133,Z 123.833,A -85,B 0,C 180,E1 -2923.735,E2 -2923.735} C_VEL
LIN {X 0,Y 559.138,Z 123.836,A -85,B 0,C 180,E1 -2926.805,E2 -2926.805} C_VEL
LIN {X 0,Y 559.149,Z 123.83,A -85,B 0,C 180,E1 -2929.189,E2 -2929.189} C_VEL
LIN {X 0,Y 559.128,Z 123.838,A -85,B 0,C 180,E1 -2931.983,E2 -2931.983} C_VEL
LIN {X 0,Y 559.127,Z 123.834,A -85,B 0,C 180,E1 -2934.788,E2 -2934.788} C_VEL
LIN {X 0,Y 559.153,Z 123.83,A -85,B 0,C 180,E1 -2937.365,E2 -2937.365} C_VEL
LIN {X 0,Y 559.146,Z 123.839,A -85,B 0,C 180,E1 -2940.144,E2 -2940.144} C_VEL
LIN {X 0,Y 559.167,Z 123.828,A -85,B 0,C 180,E1 -2943.099,E2 -2943.099} C_VEL
LIN {X 0,Y 559.198,Z 124.024,A -85,B 0,C 180,E1 -2945.893,E2 -2945.893} C_VEL
LIN {X 0,Y 560.148,Z 129.606,A -85,B 0,C 180,E1 -2946.737,E2 -2946.737} C_VEL
LIN {X 0,Y 559.87,Z 149.834,A -85,B 0,C 180,E1 -2949.615,E2 -2949.615} C_VEL
LIN {X 0,Y 559.623,Z 168.8,A -85,B 0,C 180,E1 -2952.27,E2 -2952.27} C_VEL
LIN {X 0,Y 559.413,Z 187.715,A -85,B 0,C 180,E1 -2954.89,E2 -2954.89} C_VEL
LIN {X 0,Y 559.413,Z 194.292,A -85,B 0,C 180,E1 -2955.797,E2 -2955.797} C_VEL
LIN {X 0,Y 560.298,Z 202.236,A -85,B 0,C 180,E1 -2955.936,E2 -2955.936} C_VEL
LIN {X 0,Y 560.023,Z 302.987,A -85,B 0,C 180,E1 -2957.245,E2 -2957.245} C_VEL
LIN {X 0,Y 559.899,Z 316.245,A -85,B 0,C 180,E1 -2957.565,E2 -2957.565} C_VEL
LIN {X 0,Y 559.775,Z 329.517,A -85,B 0,C 180,E1 -2958.045,E2 -2958.045} C_VEL
LIN {X 0,Y 559.65,Z 341.91,A -85,B 0,C 180,E1 -2958.667,E2 -2958.667} C_VEL
LIN {X 0,Y 559.426,Z 353.496,A -85,B 0,C 180,E1 -2959.414,E2 -2959.414} C_VEL
LIN {X 0,Y 559.296,Z 363.655,A -85,B 0,C 180,E1 -2960.234,E2 -2960.234} C_VEL
LIN {X 0,Y 559.134,Z 372.793,A -85,B 0,C 180,E1 -2961.143,E2 -2961.143} C_VEL
LIN {X 0,Y 559.009,Z 381.694,A -85,B 0,C 180,E1 -2962.233,E2 -2962.233} C_VEL
LIN {X 0,Y 558.924,Z 387.744,A -85,B 0,C 180,E1 -2963.141,E2 -2963.141} C_VEL
LIN {X 0,Y 558.935,Z 393.683,A -85,B 0,C 180,E1 -2964.228,E2 -2964.228} C_VEL
LIN {X 0,Y 558.826,Z 398.376,A -85,B 0,C 180,E1 -2965.312,E2 -2965.312} C_VEL
LIN {X 0,Y 558.836,Z 401.96,A -85,B 0,C 180,E1 -2966.396,E2 -2966.396} C_VEL
LIN {X 0,Y 558.799,Z 403.809,A -85,B 0,C 180,E1 -2967.117,E2 -2967.117} C_VEL
LIN {X 0,Y 558.745,Z 406.184,A -85,B 0,C 180,E1 -2968.559,E2 -2968.559} C_VEL
LIN {X 0,Y 558.74,Z 407,A -85,B 0,C 180,E1 -2970.001,E2 -2970.001} C_VEL
LIN {X 0,Y 558.745,Z 406.183,A -85,B 0,C 180,E1 -2971.442,E2 -2971.442} C_VEL
LIN {X 0,Y 558.799,Z 403.809,A -85,B 0,C 180,E1 -2972.884,E2 -2972.884} C_VEL
LIN {X 0,Y 558.844,Z 400.893,A -85,B 0,C 180,E1 -2973.967,E2 -2973.967} C_VEL
LIN {X 0,Y 558.798,Z 396.946,A -85,B 0,C 180,E1 -2975.051,E2 -2975.051} C_VEL
LIN {X 0,Y 558.922,Z 391.864,A -85,B 0,C 180,E1 -2976.136,E2 -2976.136} C_VEL
LIN {X 0,Y 558.978,Z 385.463,A -85,B 0,C 180,E1 -2977.223,E2 -2977.223} C_VEL
LIN {X 0,Y 559.099,Z 377.473,A -85,B 0,C 180,E1 -2978.312,E2 -2978.312} C_VEL
LIN {X 0,Y 559.195,Z 369.328,A -85,B 0,C 180,E1 -2979.222,E2 -2979.222} C_VEL
LIN {X 0,Y 559.357,Z 359.391,A -85,B 0,C 180,E1 -2980.132,E2 -2980.132} C_VEL
LIN {X 0,Y 559.556,Z 348.389,A -85,B 0,C 180,E1 -2980.937,E2 -2980.937} C_VEL
LIN {X 0,Y 559.672,Z 336.447,A -85,B 0,C 180,E1 -2981.628,E2 -2981.628} C_VEL
LIN {X 0,Y 559.797,Z 324.963,A -85,B 0,C 180,E1 -2982.14,E2 -2982.14} C_VEL
LIN {X 0,Y 559.969,Z 312.153,A -85,B 0,C 180,E1 -2982.55,E2 -2982.55} C_VEL
LIN {X 0,Y 560.091,Z 298.561,A -85,B 0,C 180,E1 -2982.824,E2 -2982.824} C_VEL
LIN {X 0,Y 560.225,Z 200.108,A -85,B 0,C 180,E1 -2984.094,E2 -2984.094} C_VEL
LIN {X 0,Y 559.413,Z 194.276,A -85,B 0,C 180,E1 -2984.204,E2 -2984.204} C_VEL
LIN {X 0,Y 559.622,Z 172.267,A -85,B 0,C 180,E1 -2987.244,E2 -2987.244} C_VEL
LIN {X 0,Y 559.873,Z 149.786,A -85,B 0,C 180,E1 -2990.386,E2 -2990.386} C_VEL
LIN {X 0,Y 560.114,Z 130.861,A -85,B 0,C 180,E1 -2993.075,E2 -2993.075} C_VEL
LIN {X 0,Y 559.456,Z 125.312,A -85,B 0,C 180,E1 -2993.9,E2 -2993.9} C_VEL
LIN {X 0,Y 559.183,Z 123.835,A -85,B 0,C 180,E1 -2994.158,E2 -2994.158} C_VEL
LIN {X 0,Y 559.161,Z 123.83,A -85,B 0,C 180,E1 -2996.903,E2 -2996.903} C_VEL
LIN {X 0,Y 559.141,Z 123.841,A -85,B 0,C 180,E1 -2999.856,E2 -2999.856} C_VEL
LIN {X 0,Y 559.158,Z 123.83,A -85,B 0,C 180,E1 -3002.715,E2 -3002.715} C_VEL
LIN {X 0,Y 559.125,Z 123.836,A -85,B 0,C 180,E1 -3005.324,E2 -3005.324} C_VEL
LIN {X 0,Y 559.132,Z 123.836,A -85,B 0,C 180,E1 -3008.018,E2 -3008.018} C_VEL
LIN {X 0,Y 559.156,Z 123.829,A -85,B 0,C 180,E1 -3010.813,E2 -3010.813} C_VEL
LIN {X 0,Y 559.137,Z 123.837,A -85,B 0,C 180,E1 -3013.734,E2 -3013.734} C_VEL
LIN {X 0,Y 559.132,Z 123.834,A -85,B 0,C 180,E1 -3016.805,E2 -3016.805} C_VEL
LIN {X 0,Y 559.154,Z 123.837,A -85,B 0,C 180,E1 -3019.187,E2 -3019.187} C_VEL
LIN {X 0,Y 559.129,Z 123.833,A -85,B 0,C 180,E1 -3021.982,E2 -3021.982} C_VEL
LIN {X 0,Y 559.127,Z 123.837,A -85,B 0,C 180,E1 -3024.788,E2 -3024.788} C_VEL
LIN {X 0,Y 559.148,Z 123.835,A -85,B 0,C 180,E1 -3027.366,E2 -3027.366} C_VEL
LIN {X 0,Y 559.11,Z 123.835,A -85,B 0,C 180,E1 -3030.15,E2 -3030.15} C_VEL
LIN {X 0,Y 559.124,Z 123.837,A -85,B 0,C 180,E1 -3033.182,E2 -3033.182} C_VEL
LIN {X 0,Y 559.112,Z 123.835,A -85,B 0,C 180,E1 -3035.493,E2 -3035.493} C_VEL
LIN {X 0,Y 559.158,Z 123.838,A -85,B 0,C 180,E1 -3038.623,E2 -3038.623} C_VEL
LIN {X 0,Y 559.151,Z 123.833,A -85,B 0,C 180,E1 -3040.926,E2 -3040.926} C_VEL
LIN {X 0,Y 559.125,Z 123.835,A -85,B 0,C 180,E1 -3043.947,E2 -3043.947} C_VEL
LIN {X 0,Y 559.138,Z 123.836,A -85,B 0,C 180,E1 -3046.183,E2 -3046.183} C_VEL
LIN {X 0,Y 559.16,Z 123.829,A -85,B 0,C 180,E1 -3049.133,E2 -3049.133} C_VEL
LIN {X 0,Y 559.131,Z 123.838,A -85,B 0,C 180,E1 -3052.053,E2 -3052.053} C_VEL
LIN {X 0,Y 559.219,Z 123.821,A -85,B 0,C 180,E1 -3054.953,E2 -3054.953} C_VEL
LIN {X 0,Y 559.246,Z 123.823,A -85,B 0,C 180,E1 -3057.839,E2 -3057.839} C_VEL
LIN {X 0,Y 559.252,Z 123.825,A -85,B 0,C 180,E1 -3060,E2 -3060} C_VEL
LIN {X 0,Y 559.205,Z 123.821,A -85,B 0,C 180,E1 -3062.882,E2 -3062.882} C_VEL
LIN {X 0,Y 559.206,Z 123.831,A -85,B 0,C 180,E1 -3065.771,E2 -3065.771} C_VEL
LIN {X 0,Y 559.158,Z 123.827,A -85,B 0,C 180,E1 -3068.675,E2 -3068.675} C_VEL
LIN {X 0,Y 559.196,Z 123.832,A -85,B 0,C 180,E1 -3071.601,E2 -3071.601} C_VEL
LIN {X 0,Y 559.157,Z 123.827,A -85,B 0,C 180,E1 -3074.578,E2 -3074.578} C_VEL
LIN {X 0,Y 559.13,Z 123.837,A -85,B 0,C 180,E1 -3077.558,E2 -3077.558} C_VEL
LIN {X 0,Y 559.162,Z 123.829,A -85,B 0,C 180,E1 -3079.838,E2 -3079.838} C_VEL
LIN {X 0,Y 559.131,Z 123.832,A -85,B 0,C 180,E1 -3082.153,E2 -3082.153} C_VEL
LIN {X 0,Y 559.139,Z 123.838,A -85,B 0,C 180,E1 -3085.178,E2 -3085.178} C_VEL
LIN {X 0,Y 559.138,Z 123.831,A -85,B 0,C 180,E1 -3087.715,E2 -3087.715} C_VEL
LIN {X 0,Y 559.129,Z 123.834,A -85,B 0,C 180,E1 -3090.574,E2 -3090.574} C_VEL
LIN {X 0,Y 558.47,Z 123.92,A -85,B 0,C 180,E1 -3091.176,E2 -3091.176} C_VEL
LIN {X 0,Y 555.612,Z 124.274,A -85,B 0,C 180,E1 -3092.152,E2 -3092.152} C_VEL
LIN {X 0,Y 553.196,Z 124.578,A -85,B 0,C 180,E1 -3092.938,E2 -3092.938} C_VEL
LIN {X 0,Y 552.168,Z 124.7,A -85,B 0,C 180,E1 -3093.544,E2 -3093.544} C_VEL
LIN {X 0,Y 552.089,Z 124.709,A -85,B 0,C 180,E1 -3093.75,E2 -3093.75} C_VEL
LIN {X 0,Y 552.107,Z 124.715,A -85,B 0,C 180,E1 -3096.747,E2 -3096.747} C_VEL
LIN {X 0,Y 552.13,Z 124.703,A -85,B 0,C 180,E1 -3099.528,E2 -3099.528} C_VEL
LIN {X 0,Y 552.132,Z 124.71,A -85,B 0,C 180,E1 -3102.426,E2 -3102.426} C_VEL
LIN {X 0,Y 552.096,Z 124.709,A -85,B 0,C 180,E1 -3105.562,E2 -3105.562} C_VEL
LIN {X 0,Y 552.123,Z 124.708,A -85,B 0,C 180,E1 -3108.679,E2 -3108.679} C_VEL
LIN {X 0,Y 552.122,Z 124.706,A -85,B 0,C 180,E1 -3111.411,E2 -3111.411} C_VEL
LIN {X 0,Y 552.089,Z 124.718,A -85,B 0,C 180,E1 -3114.156,E2 -3114.156} C_VEL
LIN {X 0,Y 552.119,Z 124.706,A -85,B 0,C 180,E1 -3116.814,E2 -3116.814} C_VEL
LIN {X 0,Y 552.106,Z 124.711,A -85,B 0,C 180,E1 -3119.391,E2 -3119.391} C_VEL
LIN {X 0,Y 552.095,Z 124.717,A -85,B 0,C 180,E1 -3121.901,E2 -3121.901} C_VEL
LIN {X 0,Y 552.161,Z 124.703,A -85,B 0,C 180,E1 -3124.65,E2 -3124.65} C_VEL
LIN {X 0,Y 552.171,Z 124.872,A -85,B 0,C 180,E1 -3126.459,E2 -3126.459} C_VEL
LIN {X 0,Y 552.389,Z 130.637,A -85,B 0,C 180,E1 -3127.561,E2 -3127.561} C_VEL
LIN {X 0,Y 552.231,Z 145.377,A -85,B 0,C 180,E1 -3130.351,E2 -3130.351} C_VEL
LIN {X 0,Y 552.216,Z 147.099,A -85,B 0,C 180,E1 -3130.676,E2 -3130.676} C_VEL
LIN {X 0,Y 553.408,Z 154.051,A -85,B 0,C 180,E1 -3130.816,E2 -3130.816} C_VEL
LIN {X 0,Y 553.118,Z 253.313,A -85,B 0,C 180,E1 -3132.125,E2 -3132.125} C_VEL
LIN {X 0,Y 552.938,Z 266.805,A -85,B 0,C 180,E1 -3132.454,E2 -3132.454} C_VEL
LIN {X 0,Y 552.854,Z 279.823,A -85,B 0,C 180,E1 -3132.933,E2 -3132.933} C_VEL
LIN {X 0,Y 552.709,Z 290.638,A -85,B 0,C 180,E1 -3133.47,E2 -3133.47} C_VEL
LIN {X 0,Y 552.507,Z 301.11,A -85,B 0,C 180,E1 -3134.128,E2 -3134.128} C_VEL
LIN {X 0,Y 552.324,Z 311.883,A -85,B 0,C 180,E1 -3134.973,E2 -3134.973} C_VEL
LIN {X 0,Y 552.175,Z 320.82,A -85,B 0,C 180,E1 -3135.835,E2 -3135.835} C_VEL
LIN {X 0,Y 552.004,Z 328.675,A -85,B 0,C 180,E1 -3136.751,E2 -3136.751} C_VEL
LIN {X 0,Y 551.921,Z 336.492,A -85,B 0,C 180,E1 -3137.871,E2 -3137.871} C_VEL
LIN {X 0,Y 551.805,Z 342.714,A -85,B 0,C 180,E1 -3138.986,E2 -3138.986} C_VEL
LIN {X 0,Y 551.76,Z 347.635,A -85,B 0,C 180,E1 -3140.098,E2 -3140.098} C_VEL
LIN {X 0,Y 551.715,Z 351.417,A -85,B 0,C 180,E1 -3141.207,E2 -3141.207} C_VEL
LIN {X 0,Y 551.713,Z 353.378,A -85,B 0,C 180,E1 -3141.944,E2 -3141.944} C_VEL
LIN {X 0,Y 551.697,Z 354.917,A -85,B 0,C 180,E1 -3142.681,E2 -3142.681} C_VEL
LIN {X 0,Y 551.748,Z 356.076,A -85,B 0,C 180,E1 -3143.487,E2 -3143.487} C_VEL
LIN {X 0,Y 551.681,Z 356.971,A -85,B 0,C 180,E1 -3144.883,E2 -3144.883} C_VEL
LIN {X 0,Y 551.699,Z 356.878,A -85,B 0,C 180,E1 -3145.616,E2 -3145.616} C_VEL
LIN {X 0,Y 551.732,Z 356.354,A -85,B 0,C 180,E1 -3146.348,E2 -3146.348} C_VEL
LIN {X 0,Y 551.719,Z 355.433,A -85,B 0,C 180,E1 -3147.079,E2 -3147.079} C_VEL
LIN {X 0,Y 551.653,Z 352.409,A -85,B 0,C 180,E1 -3148.539,E2 -3148.539} C_VEL
LIN {X 0,Y 551.747,Z 348.997,A -85,B 0,C 180,E1 -3149.634,E2 -3149.634} C_VEL
LIN {X 0,Y 551.724,Z 344.539,A -85,B 0,C 180,E1 -3150.729,E2 -3150.729} C_VEL
LIN {X 0,Y 551.886,Z 337.775,A -85,B 0,C 180,E1 -3152.006,E2 -3152.006} C_VEL
LIN {X 0,Y 552.012,Z 330.464,A -85,B 0,C 180,E1 -3153.101,E2 -3153.101} C_VEL
LIN {X 0,Y 552.147,Z 323.022,A -85,B 0,C 180,E1 -3154.014,E2 -3154.014} C_VEL
LIN {X 0,Y 552.276,Z 314.033,A -85,B 0,C 180,E1 -3154.927,E2 -3154.927} C_VEL
LIN {X 0,Y 552.46,Z 304.07,A -85,B 0,C 180,E1 -3155.749,E2 -3155.749} C_VEL
LIN {X 0,Y 552.647,Z 293.032,A -85,B 0,C 180,E1 -3156.48,E2 -3156.48} C_VEL
LIN {X 0,Y 552.832,Z 281.761,A -85,B 0,C 180,E1 -3157.068,E2 -3157.068} C_VEL
LIN {X 0,Y 552.958,Z 269.477,A -85,B 0,C 180,E1 -3157.553,E2 -3157.553} C_VEL
LIN {X 0,Y 553.067,Z 256.145,A -85,B 0,C 180,E1 -3157.908,E2 -3157.908} C_VEL
LIN {X 0,Y 553.178,Z 236.935,A -85,B 0,C 180,E1 -3158.194,E2 -3158.194} C_VEL
LIN {X 0,Y 553.332,Z 153.422,A -85,B 0,C 180,E1 -3159.284,E2 -3159.284} C_VEL
LIN {X 0,Y 552.197,Z 147.135,A -85,B 0,C 180,E1 -3159.407,E2 -3159.407} C_VEL
LIN {X 0,Y 552.345,Z 132.844,A -85,B 0,C 180,E1 -3162.118,E2 -3162.118} C_VEL
LIN {X 0,Y 552.176,Z 124.989,A -85,B 0,C 180,E1 -3163.618,E2 -3163.618} C_VEL
LIN {X 0,Y 552.145,Z 124.709,A -85,B 0,C 180,E1 -3163.807,E2 -3163.807} C_VEL
LIN {X 0,Y 552.135,Z 124.706,A -85,B 0,C 180,E1 -3167.022,E2 -3167.022} C_VEL
LIN {X 0,Y 552.127,Z 124.712,A -85,B 0,C 180,E1 -3170.1,E2 -3170.1} C_VEL
LIN {X 0,Y 552.092,Z 124.714,A -85,B 0,C 180,E1 -3172.45,E2 -3172.45} C_VEL
LIN {X 0,Y 552.156,Z 124.702,A -85,B 0,C 180,E1 -3175.349,E2 -3175.349} C_VEL
LIN {X 0,Y 552.088,Z 124.718,A -85,B 0,C 180,E1 -3178.098,E2 -3178.098} C_VEL
LIN {X 0,Y 552.101,Z 124.709,A -85,B 0,C 180,E1 -3180.608,E2 -3180.608} C_VEL
LIN {X 0,Y 552.112,Z 124.708,A -85,B 0,C 180,E1 -3183.185,E2 -3183.185} C_VEL
LIN {X 0,Y 552.082,Z 124.719,A -85,B 0,C 180,E1 -3185.843,E2 -3185.843} C_VEL
LIN {X 0,Y 552.12,Z 124.708,A -85,B 0,C 180,E1 -3189.06,E2 -3189.06} C_VEL
LIN {X 0,Y 552.115,Z 124.713,A -85,B 0,C 180,E1 -3191.445,E2 -3191.445} C_VEL
LIN {X 0,Y 552.084,Z 124.711,A -85,B 0,C 180,E1 -3194.53,E2 -3194.53} C_VEL
LIN {X 0,Y 552.122,Z 124.712,A -85,B 0,C 180,E1 -3197.584,E2 -3197.584} C_VEL
LIN {X 0,Y 552.12,Z 124.707,A -85,B 0,C 180,E1 -3200.472,E2 -3200.472} C_VEL
LIN {X 0,Y 552.098,Z 124.717,A -85,B 0,C 180,E1 -3203.316,E2 -3203.316} C_VEL
LIN {X 0,Y 552.092,Z 124.71,A -85,B 0,C 180,E1 -3205.936,E2 -3205.936} C_VEL
LIN {X 0,Y 552.11,Z 124.711,A -85,B 0,C 180,E1 -3208.54,E2 -3208.54} C_VEL
LIN {X 0,Y 552.094,Z 124.712,A -85,B 0,C 180,E1 -3211.441,E2 -3211.441} C_VEL
LIN {X 0,Y 552.094,Z 124.711,A -85,B 0,C 180,E1 -3213.542,E2 -3213.542} C_VEL
LIN {X 0,Y 552.077,Z 124.719,A -85,B 0,C 180,E1 -3216.757,E2 -3216.757} C_VEL
LIN {X 0,Y 552.103,Z 124.712,A -85,B 0,C 180,E1 -3219.119,E2 -3219.119} C_VEL
LIN {X 0,Y 552.07,Z 124.713,A -85,B 0,C 180,E1 -3221.442,E2 -3221.442} C_VEL
LIN {X 0,Y 552.07,Z 124.713,A -85,B 0,C 180,E1 -3223.736,E2 -3223.736} C_VEL
LIN {X 0,Y 552.099,Z 124.712,A -85,B 0,C 180,E1 -3226.003,E2 -3226.003} C_VEL
LIN {X 0,Y 552.146,Z 124.705,A -85,B 0,C 180,E1 -3228.993,E2 -3228.993} C_VEL
LIN {X 0,Y 552.129,Z 124.711,A -85,B 0,C 180,E1 -3231.951,E2 -3231.951} C_VEL
LIN {X 0,Y 552.195,Z 124.698,A -85,B 0,C 180,E1 -3234.889,E2 -3234.889} C_VEL
LIN {X 0,Y 552.209,Z 124.701,A -85,B 0,C 180,E1 -3237.812,E2 -3237.812} C_VEL
LIN {X 0,Y 552.21,Z 124.702,A -85,B 0,C 180,E1 -3240,E2 -3240} C_VEL
LIN {X 0,Y 552.164,Z 124.701,A -85,B 0,C 180,E1 -3242.918,E2 -3242.918} C_VEL
LIN {X 0,Y 552.174,Z 124.707,A -85,B 0,C 180,E1 -3245.844,E2 -3245.844} C_VEL
LIN {X 0,Y 552.12,Z 124.707,A -85,B 0,C 180,E1 -3248.786,E2 -3248.786} C_VEL
LIN {X 0,Y 552.143,Z 124.71,A -85,B 0,C 180,E1 -3251.751,E2 -3251.751} C_VEL
LIN {X 0,Y 552.108,Z 124.709,A -85,B 0,C 180,E1 -3254.749,E2 -3254.749} C_VEL
LIN {X 0,Y 552.076,Z 124.716,A -85,B 0,C 180,E1 -3257.79,E2 -3257.79} C_VEL
LIN {X 0,Y 552.111,Z 124.708,A -85,B 0,C 180,E1 -3260.102,E2 -3260.102} C_VEL
LIN {X 0,Y 552.074,Z 124.713,A -85,B 0,C 180,E1 -3262.452,E2 -3262.452} C_VEL
LIN {X 0,Y 552.096,Z 124.712,A -85,B 0,C 180,E1 -3265.646,E2 -3265.646} C_VEL
LIN {X 0,Y 552.082,Z 124.711,A -85,B 0,C 180,E1 -3268.1,E2 -3268.1} C_VEL
LIN {X 0,Y 552.09,Z 124.714,A -85,B 0,C 180,E1 -3270.61,E2 -3270.61} C_VEL
LIN {X 0,Y 552.096,Z 124.714,A -85,B 0,C 180,E1 -3273.187,E2 -3273.187} C_VEL
LIN {X 0,Y 552.076,Z 124.712,A -85,B 0,C 180,E1 -3275.844,E2 -3275.844} C_VEL
LIN {X 0,Y 552.112,Z 124.711,A -85,B 0,C 180,E1 -3279.062,E2 -3279.062} C_VEL
LIN {X 0,Y 552.112,Z 124.707,A -85,B 0,C 180,E1 -3281.447,E2 -3281.447} C_VEL
LIN {X 0,Y 552.086,Z 124.718,A -85,B 0,C 180,E1 -3284.533,E2 -3284.533} C_VEL
LIN {X 0,Y 552.123,Z 124.706,A -85,B 0,C 180,E1 -3287.586,E2 -3287.586} C_VEL
LIN {X 0,Y 552.127,Z 124.712,A -85,B 0,C 180,E1 -3290.474,E2 -3290.474} C_VEL
LIN {X 0,Y 552.101,Z 124.708,A -85,B 0,C 180,E1 -3293.318,E2 -3293.318} C_VEL
LIN {X 0,Y 552.122,Z 124.711,A -85,B 0,C 180,E1 -3295.94,E2 -3295.94} C_VEL
LIN {X 0,Y 552.116,Z 124.709,A -85,B 0,C 180,E1 -3298.542,E2 -3298.542} C_VEL
LIN {X 0,Y 552.121,Z 124.709,A -85,B 0,C 180,E1 -3301.439,E2 -3301.439} C_VEL
LIN {X 0,Y 552.128,Z 124.707,A -85,B 0,C 180,E1 -3304.357,E2 -3304.357} C_VEL
LIN {X 0,Y 552.143,Z 124.732,A -85,B 0,C 180,E1 -3305.715,E2 -3305.715} C_VEL
LIN {X 0,Y 553.144,Z 130.08,A -85,B 0,C 180,E1 -3306.539,E2 -3306.539} C_VEL
LIN {X 0,Y 552.965,Z 145.457,A -85,B 0,C 180,E1 -3308.764,E2 -3308.764} C_VEL
LIN {X 0,Y 552.711,Z 165.781,A -85,B 0,C 180,E1 -3311.658,E2 -3311.658} C_VEL
LIN {X 0,Y 552.436,Z 184.702,A -85,B 0,C 180,E1 -3314.317,E2 -3314.317} C_VEL
LIN {X 0,Y 552.369,Z 194.072,A -85,B 0,C 180,E1 -3315.626,E2 -3315.626} C_VEL
LIN {X 0,Y 553.423,Z 202.369,A -85,B 0,C 180,E1 -3315.763,E2 -3315.763} C_VEL
LIN {X 0,Y 553.1,Z 302.659,A -85,B 0,C 180,E1 -3317.083,E2 -3317.083} C_VEL
LIN {X 0,Y 552.966,Z 315.945,A -85,B 0,C 180,E1 -3317.406,E2 -3317.406} C_VEL
LIN {X 0,Y 552.794,Z 329.251,A -85,B 0,C 180,E1 -3317.892,E2 -3317.892} C_VEL
LIN {X 0,Y 552.638,Z 341.766,A -85,B 0,C 180,E1 -3318.525,E2 -3318.525} C_VEL
LIN {X 0,Y 552.428,Z 353.348,A -85,B 0,C 180,E1 -3319.278,E2 -3319.278} C_VEL
LIN {X 0,Y 552.282,Z 363.569,A -85,B 0,C 180,E1 -3320.109,E2 -3320.109} C_VEL
LIN {X 0,Y 552.103,Z 372.767,A -85,B 0,C 180,E1 -3321.03,E2 -3321.03} C_VEL
LIN {X 0,Y 551.959,Z 381.693,A -85,B 0,C 180,E1 -3322.134,E2 -3322.134} C_VEL
LIN {X 0,Y 551.834,Z 388.853,A -85,B 0,C 180,E1 -3323.235,E2 -3323.235} C_VEL
LIN {X 0,Y 551.804,Z 395.369,A -85,B 0,C 180,E1 -3324.519,E2 -3324.519} C_VEL
LIN {X 0,Y 551.764,Z 399.679,A -85,B 0,C 180,E1 -3325.618,E2 -3325.618} C_VEL
LIN {X 0,Y 551.75,Z 401.96,A -85,B 0,C 180,E1 -3326.349,E2 -3326.349} C_VEL
LIN {X 0,Y 551.723,Z 403.808,A -85,B 0,C 180,E1 -3327.08,E2 -3327.08} C_VEL
LIN {X 0,Y 551.645,Z 406.183,A -85,B 0,C 180,E1 -3328.541,E2 -3328.541} C_VEL
LIN {X 0,Y 551.64,Z 407,A -85,B 0,C 180,E1 -3330.001,E2 -3330.001} C_VEL
LIN {X 0,Y 551.645,Z 406.183,A -85,B 0,C 180,E1 -3331.461,E2 -3331.461} C_VEL
LIN {X 0,Y 551.723,Z 403.809,A -85,B 0,C 180,E1 -3332.921,E2 -3332.921} C_VEL
LIN {X 0,Y 551.764,Z 400.893,A -85,B 0,C 180,E1 -3334.018,E2 -3334.018} C_VEL
LIN {X 0,Y 551.724,Z 396.946,A -85,B 0,C 180,E1 -3335.116,E2 -3335.116} C_VEL
LIN {X 0,Y 551.803,Z 391.187,A -85,B 0,C 180,E1 -3336.342,E2 -3336.342} C_VEL
LIN {X 0,Y 551.927,Z 384.231,A -85,B 0,C 180,E1 -3337.5,E2 -3337.5} C_VEL
LIN {X 0,Y 552.083,Z 375.982,A -85,B 0,C 180,E1 -3338.603,E2 -3338.603} C_VEL
LIN {X 0,Y 552.201,Z 367.472,A -85,B 0,C 180,E1 -3339.524,E2 -3339.524} C_VEL
LIN {X 0,Y 552.413,Z 356.957,A -85,B 0,C 180,E1 -3340.446,E2 -3340.446} C_VEL
LIN {X 0,Y 552.556,Z 346.09,A -85,B 0,C 180,E1 -3341.215,E2 -3341.215} C_VEL
LIN {X 0,Y 552.753,Z 335.158,A -85,B 0,C 180,E1 -3341.831,E2 -3341.831} C_VEL
LIN {X 0,Y 552.903,Z 323.468,A -85,B 0,C 180,E1 -3342.34,E2 -3342.34} C_VEL
LIN {X 0,Y 553.051,Z 310.004,A -85,B 0,C 180,E1 -3342.756,E2 -3342.756} C_VEL
LIN {X 0,Y 553.176,Z 296.702,A -85,B 0,C 180,E1 -3343.01,E2 -3343.01} C_VEL
LIN {X 0,Y 553.244,Z 200.251,A -85,B 0,C 180,E1 -3344.269,E2 -3344.269} C_VEL
LIN {X 0,Y 552.38,Z 193.925,A -85,B 0,C 180,E1 -3344.392,E2 -3344.392} C_VEL
LIN {X 0,Y 552.592,Z 171.936,A -85,B 0,C 180,E1 -3347.47,E2 -3347.47} C_VEL
LIN {X 0,Y 552.906,Z 150.823,A -85,B 0,C 180,E1 -3350.46,E2 -3350.46} C_VEL
LIN {X 0,Y 553.164,Z 131.823,A -85,B 0,C 180,E1 -3353.195,E2 -3353.195} C_VEL
LIN {X 0,Y 552.453,Z 126.346,A -85,B 0,C 180,E1 -3354.022,E2 -3354.022} C_VEL
LIN {X 0,Y 552.129,Z 124.713,A -85,B 0,C 180,E1 -3354.287,E2 -3354.287} C_VEL
LIN {X 0,Y 552.1,Z 124.711,A -85,B 0,C 180,E1 -3357.276,E2 -3357.276} C_VEL
LIN {X 0,Y 552.111,Z 124.717,A -85,B 0,C 180,E1 -3360.049,E2 -3360.049} C_VEL
LIN {X 0,Y 552.117,Z 124.707,A -85,B 0,C 180,E1 -3362.846,E2 -3362.846} C_VEL
LIN {X 0,Y 552.073,Z 124.716,A -85,B 0,C 180,E1 -3365.439,E2 -3365.439} C_VEL
LIN {X 0,Y 552.096,Z 124.715,A -85,B 0,C 180,E1 -3367.885,E2 -3367.885} C_VEL
LIN {X 0,Y 552.11,Z 124.707,A -85,B 0,C 180,E1 -3370.481,E2 -3370.481} C_VEL
LIN {X 0,Y 552.094,Z 124.718,A -85,B 0,C 180,E1 -3373.482,E2 -3373.482} C_VEL
LIN {X 0,Y 552.073,Z 124.712,A -85,B 0,C 180,E1 -3376.573,E2 -3376.573} C_VEL
LIN {X 0,Y 552.107,Z 124.713,A -85,B 0,C 180,E1 -3379.519,E2 -3379.519} C_VEL
LIN {X 0,Y 552.09,Z 124.71,A -85,B 0,C 180,E1 -3382.336,E2 -3382.336} C_VEL
LIN {X 0,Y 552.079,Z 124.72,A -85,B 0,C 180,E1 -3385.05,E2 -3385.05} C_VEL
LIN {X 0,Y 552.107,Z 124.709,A -85,B 0,C 180,E1 -3387.681,E2 -3387.681} C_VEL
LIN {X 0,Y 552.075,Z 124.712,A -85,B 0,C 180,E1 -3390.233,E2 -3390.233} C_VEL
LIN {X 0,Y 552.092,Z 124.715,A -85,B 0,C 180,E1 -3393.009,E2 -3393.009} C_VEL
LIN {X 0,Y 552.075,Z 124.712,A -85,B 0,C 180,E1 -3395.961,E2 -3395.961} C_VEL
LIN {X 0,Y 552.094,Z 124.71,A -85,B 0,C 180,E1 -3399.119,E2 -3399.119} C_VEL
LIN {X 0,Y 552.074,Z 124.71,A -85,B 0,C 180,E1 -3401.443,E2 -3401.443} C_VEL
LIN {X 0,Y 552.069,Z 124.712,A -85,B 0,C 180,E1 -3403.736,E2 -3403.736} C_VEL
LIN {X 0,Y 552.1,Z 124.71,A -85,B 0,C 180,E1 -3406.004,E2 -3406.004} C_VEL
LIN {X 0,Y 552.122,Z 124.706,A -85,B 0,C 180,E1 -3408.993,E2 -3408.993} C_VEL
LIN {X 0,Y 552.101,Z 124.712,A -85,B 0,C 180,E1 -3411.951,E2 -3411.951} C_VEL
LIN {X 0,Y 552.197,Z 124.696,A -85,B 0,C 180,E1 -3414.889,E2 -3414.889} C_VEL
LIN {X 0,Y 552.217,Z 124.698,A -85,B 0,C 180,E1 -3417.812,E2 -3417.812} C_VEL
LIN {X 0,Y 552.22,Z 124.701,A -85,B 0,C 180,E1 -3420,E2 -3420} C_VEL
LIN {X 0,Y 552.173,Z 124.697,A -85,B 0,C 180,E1 -3422.918,E2 -3422.918} C_VEL
LIN {X 0,Y 552.174,Z 124.706,A -85,B 0,C 180,E1 -3425.844,E2 -3425.844} C_VEL
LIN {X 0,Y 552.13,Z 124.702,A -85,B 0,C 180,E1 -3428.786,E2 -3428.786} C_VEL
LIN {X 0,Y 552.151,Z 124.707,A -85,B 0,C 180,E1 -3431.751,E2 -3431.751} C_VEL
LIN {X 0,Y 552.12,Z 124.705,A -85,B 0,C 180,E1 -3434.749,E2 -3434.749} C_VEL
LIN {X 0,Y 552.088,Z 124.711,A -85,B 0,C 180,E1 -3437.789,E2 -3437.789} C_VEL
LIN {X 0,Y 552.123,Z 124.704,A -85,B 0,C 180,E1 -3440.102,E2 -3440.102} C_VEL
LIN {X 0,Y 552.083,Z 124.711,A -85,B 0,C 180,E1 -3442.452,E2 -3442.452} C_VEL
LIN {X 0,Y 552.083,Z 124.715,A -85,B 0,C 180,E1 -3445.334,E2 -3445.334} C_VEL
LIN {X 0,Y 552.088,Z 124.709,A -85,B 0,C 180,E1 -3448.1,E2 -3448.1} C_VEL
LIN {X 0,Y 552.094,Z 124.714,A -85,B 0,C 180,E1 -3450.61,E2 -3450.61} C_VEL
LIN {X 0,Y 552.107,Z 124.71,A -85,B 0,C 180,E1 -3453.187,E2 -3453.187} C_VEL
LIN {X 0,Y 552.089,Z 124.709,A -85,B 0,C 180,E1 -3453.75,E2 -3453.75} C_VEL
LIN {X 0,Y 551.448,Z 124.794,A -85,B 0,C 180,E1 -3454.358,E2 -3454.358} C_VEL
LIN {X 0,Y 548.639,Z 125.147,A -85,B 0,C 180,E1 -3455.347,E2 -3455.347} C_VEL
LIN {X 0,Y 546.234,Z 125.449,A -85,B 0,C 180,E1 -3456.143,E2 -3456.143} C_VEL
LIN {X 0,Y 545.17,Z 125.579,A -85,B 0,C 180,E1 -3456.756,E2 -3456.756} C_VEL
LIN {X 0,Y 545.067,Z 125.588,A -85,B 0,C 180,E1 -3456.964,E2 -3456.964} C_VEL
LIN {X 0,Y 545.066,Z 125.587,A -85,B 0,C 180,E1 -3460.143,E2 -3460.143} C_VEL
LIN {X 0,Y 545.081,Z 125.583,A -85,B 0,C 180,E1 -3463.107,E2 -3463.107} C_VEL
LIN {X 0,Y 545.052,Z 125.594,A -85,B 0,C 180,E1 -3466.226,E2 -3466.226} C_VEL
LIN {X 0,Y 545.084,Z 125.584,A -85,B 0,C 180,E1 -3468.885,E2 -3468.885} C_VEL
LIN {X 0,Y 545.086,Z 125.583,A -85,B 0,C 180,E1 -3470.819,E2 -3470.819} C_VEL
LIN {X 0,Y 545.045,Z 125.59,A -85,B 0,C 180,E1 -3473.62,E2 -3473.62} C_VEL
LIN {X 0,Y 545.069,Z 125.588,A -85,B 0,C 180,E1 -3476.328,E2 -3476.328} C_VEL
LIN {X 0,Y 545.07,Z 125.584,A -85,B 0,C 180,E1 -3478.952,E2 -3478.952} C_VEL
LIN {X 0,Y 545.087,Z 125.588,A -85,B 0,C 180,E1 -3481.507,E2 -3481.507} C_VEL
LIN {X 0,Y 545.1,Z 125.583,A -85,B 0,C 180,E1 -3484.491,E2 -3484.491} C_VEL
LIN {X 0,Y 545.142,Z 125.603,A -85,B 0,C 180,E1 -3486.343,E2 -3486.343} C_VEL
LIN {X 0,Y 545.401,Z 131.391,A -85,B 0,C 180,E1 -3487.458,E2 -3487.458} C_VEL
LIN {X 0,Y 545.22,Z 147.342,A -85,B 0,C 180,E1 -3490.492,E2 -3490.492} C_VEL
LIN {X 0,Y 546.554,Z 155.489,A -85,B 0,C 180,E1 -3490.648,E2 -3490.648} C_VEL
LIN {X 0,Y 546.222,Z 253.886,A -85,B 0,C 180,E1 -3491.964,E2 -3491.964} C_VEL
LIN {X 0,Y 546.033,Z 267.269,A -85,B 0,C 180,E1 -3492.296,E2 -3492.296} C_VEL
LIN {X 0,Y 545.918,Z 280.129,A -85,B 0,C 180,E1 -3492.776,E2 -3492.776} C_VEL
LIN {X 0,Y 545.763,Z 291.45,A -85,B 0,C 180,E1 -3493.35,E2 -3493.35} C_VEL
LIN {X 0,Y 545.537,Z 301.83,A -85,B 0,C 180,E1 -3494.016,E2 -3494.016} C_VEL
LIN {X 0,Y 545.327,Z 312.534,A -85,B 0,C 180,E1 -3494.872,E2 -3494.872} C_VEL
LIN {X 0,Y 545.173,Z 322.137,A -85,B 0,C 180,E1 -3495.822,E2 -3495.822} C_VEL
LIN {X 0,Y 544.952,Z 331.312,A -85,B 0,C 180,E1 -3496.956,E2 -3496.956} C_VEL
LIN {X 0,Y 544.863,Z 338.67,A -85,B 0,C 180,E1 -3498.089,E2 -3498.089} C_VEL
LIN {X 0,Y 544.718,Z 344.536,A -85,B 0,C 180,E1 -3499.217,E2 -3499.217} C_VEL
LIN {X 0,Y 544.658,Z 349.134,A -85,B 0,C 180,E1 -3500.343,E2 -3500.343} C_VEL
LIN {X 0,Y 544.653,Z 351.554,A -85,B 0,C 180,E1 -3501.092,E2 -3501.092} C_VEL
LIN {X 0,Y 544.63,Z 353.526,A -85,B 0,C 180,E1 -3501.839,E2 -3501.839} C_VEL
LIN {X 0,Y 544.611,Z 355.083,A -85,B 0,C 180,E1 -3502.585,E2 -3502.585} C_VEL
LIN {X 0,Y 544.669,Z 356.377,A -85,B 0,C 180,E1 -3503.492,E2 -3503.492} C_VEL
LIN {X 0,Y 544.601,Z 357.225,A -85,B 0,C 180,E1 -3504.817,E2 -3504.817} C_VEL
LIN {X 0,Y 544.6,Z 357.163,A -85,B 0,C 180,E1 -3505.559,E2 -3505.559} C_VEL
LIN {X 0,Y 544.646,Z 356.694,A -85,B 0,C 180,E1 -3506.3,E2 -3506.3} C_VEL
LIN {X 0,Y 544.646,Z 355.81,A -85,B 0,C 180,E1 -3507.041,E2 -3507.041} C_VEL
LIN {X 0,Y 544.564,Z 352.883,A -85,B 0,C 180,E1 -3508.52,E2 -3508.52} C_VEL
LIN {X 0,Y 544.678,Z 349.533,A -85,B 0,C 180,E1 -3509.63,E2 -3509.63} C_VEL
LIN {X 0,Y 544.651,Z 345.14,A -85,B 0,C 180,E1 -3510.739,E2 -3510.739} C_VEL
LIN {X 0,Y 544.849,Z 338.478,A -85,B 0,C 180,E1 -3512.032,E2 -3512.032} C_VEL
LIN {X 0,Y 544.964,Z 331.251,A -85,B 0,C 180,E1 -3513.141,E2 -3513.141} C_VEL
LIN {X 0,Y 545.12,Z 323.901,A -85,B 0,C 180,E1 -3514.065,E2 -3514.065} C_VEL
LIN {X 0,Y 545.313,Z 314.052,A -85,B 0,C 180,E1 -3515.083,E2 -3515.083} C_VEL
LIN {X 0,Y 545.475,Z 304.008,A -85,B 0,C 180,E1 -3515.915,E2 -3515.915} C_VEL
LIN {X 0,Y 545.706,Z 292.878,A -85,B 0,C 180,E1 -3516.655,E2 -3516.655} C_VEL
LIN {X 0,Y 545.902,Z 281.739,A -85,B 0,C 180,E1 -3517.239,E2 -3517.239} C_VEL
LIN {X 0,Y 546.058,Z 269.489,A -85,B 0,C 180,E1 -3517.724,E2 -3517.724} C_VEL
LIN {X 0,Y 546.165,Z 256.779,A -85,B 0,C 180,E1 -3518.067,E2 -3518.067} C_VEL
LIN {X 0,Y 546.27,Z 238.632,A -85,B 0,C 180,E1 -3518.344,E2 -3518.344} C_VEL
LIN {X 0,Y 546.504,Z 154.457,A -85,B 0,C 180,E1 -3519.456,E2 -3519.456} C_VEL
LIN {X 0,Y 545.202,Z 147.359,A -85,B 0,C 180,E1 -3519.599,E2 -3519.599} C_VEL
LIN {X 0,Y 545.362,Z 133.304,A -85,B 0,C 180,E1 -3522.276,E2 -3522.276} C_VEL
LIN {X 0,Y 545.139,Z 125.891,A -85,B 0,C 180,E1 -3523.702,E2 -3523.702} C_VEL
LIN {X 0,Y 545.1,Z 125.587,A -85,B 0,C 180,E1 -3523.798,E2 -3523.798} C_VEL
LIN {X 0,Y 545.067,Z 125.593,A -85,B 0,C 180,E1 -3526.478,E2 -3526.478} C_VEL
LIN {X 0,Y 545.117,Z 125.579,A -85,B 0,C 180,E1 -3529.584,E2 -3529.584} C_VEL
LIN {X 0,Y 545.037,Z 125.59,A -85,B 0,C 180,E1 -3532.757,E2 -3532.757} C_VEL
LIN {X 0,Y 545.094,Z 125.583,A -85,B 0,C 180,E1 -3535.508,E2 -3535.508} C_VEL
LIN {X 0,Y 545.081,Z 125.585,A -85,B 0,C 180,E1 -3538.492,E2 -3538.492} C_VEL
LIN {X 0,Y 545.064,Z 125.585,A -85,B 0,C 180,E1 -3541.047,E2 -3541.047} C_VEL
LIN {X 0,Y 545.062,Z 125.591,A -85,B 0,C 180,E1 -3543.671,E2 -3543.671} C_VEL
LIN {X 0,Y 545.066,Z 125.585,A -85,B 0,C 180,E1 -3546.925,E2 -3546.925} C_VEL
LIN {X 0,Y 545.063,Z 125.587,A -85,B 0,C 180,E1 -3550.141,E2 -3550.141} C_VEL
LIN {X 0,Y 545.073,Z 125.588,A -85,B 0,C 180,E1 -3553.105,E2 -3553.105} C_VEL
LIN {X 0,Y 545.043,Z 125.588,A -85,B 0,C 180,E1 -3556.225,E2 -3556.225} C_VEL
LIN {X 0,Y 545.073,Z 125.587,A -85,B 0,C 180,E1 -3558.884,E2 -3558.884} C_VEL
LIN {X 0,Y 545.07,Z 125.588,A -85,B 0,C 180,E1 -3560.817,E2 -3560.817} C_VEL
LIN {X 0,Y 545.033,Z 125.592,A -85,B 0,C 180,E1 -3563.619,E2 -3563.619} C_VEL
LIN {X 0,Y 545.039,Z 125.589,A -85,B 0,C 180,E1 -3566.326,E2 -3566.326} C_VEL
LIN {X 0,Y 545.054,Z 125.593,A -85,B 0,C 180,E1 -3568.951,E2 -3568.951} C_VEL
LIN {X 0,Y 545.072,Z 125.586,A -85,B 0,C 180,E1 -3571.506,E2 -3571.506} C_VEL
LIN {X 0,Y 545.041,Z 125.589,A -85,B 0,C 180,E1 -3573.997,E2 -3573.997} C_VEL
LIN {X 0,Y 545.017,Z 125.594,A -85,B 0,C 180,E1 -3577.241,E2 -3577.241} C_VEL
LIN {X 0,Y 545.103,Z 125.587,A -85,B 0,C 180,E1 -3580.414,E2 -3580.414} C_VEL
LIN {X 0,Y 545.022,Z 125.591,A -85,B 0,C 180,E1 -3583.519,E2 -3583.519} C_VEL
LIN {X 0,Y 545.057,Z 125.588,A -85,B 0,C 180,E1 -3585.819,E2 -3585.819} C_VEL
LIN {X 0,Y 545.103,Z 125.583,A -85,B 0,C 180,E1 -3588.849,E2 -3588.849} C_VEL
LIN {X 0,Y 545.078,Z 125.588,A -85,B 0,C 180,E1 -3591.846,E2 -3591.846} C_VEL
LIN {X 0,Y 545.153,Z 125.576,A -85,B 0,C 180,E1 -3594.822,E2 -3594.822} C_VEL
LIN {X 0,Y 545.18,Z 125.577,A -85,B 0,C 180,E1 -3597.784,E2 -3597.784} C_VEL
LIN {X 0,Y 545.178,Z 125.578,A -85,B 0,C 180,E1 -3600,E2 -3600} C_VEL
LIN {X 0,Y 545.132,Z 125.577,A -85,B 0,C 180,E1 -3602.956,E2 -3602.956} C_VEL
LIN {X 0,Y 545.144,Z 125.582,A -85,B 0,C 180,E1 -3605.92,E2 -3605.92} C_VEL
LIN {X 0,Y 545.081,Z 125.584,A -85,B 0,C 180,E1 -3608.901,E2 -3608.901} C_VEL
LIN {X 0,Y 545.086,Z 125.588,A -85,B 0,C 180,E1 -3611.905,E2 -3611.905} C_VEL
LIN {X 0,Y 545.064,Z 125.588,A -85,B 0,C 180,E1 -3614.944,E2 -3614.944} C_VEL
LIN {X 0,Y 545.043,Z 125.59,A -85,B 0,C 180,E1 -3618.027,E2 -3618.027} C_VEL
LIN {X 0,Y 545.077,Z 125.584,A -85,B 0,C 180,E1 -3620.373,E2 -3620.373} C_VEL
LIN {X 0,Y 545.058,Z 125.59,A -85,B 0,C 180,E1 -3623.56,E2 -3623.56} C_VEL
LIN {X 0,Y 545.081,Z 125.588,A -85,B 0,C 180,E1 -3626.825,E2 -3626.825} C_VEL
LIN {X 0,Y 545.046,Z 125.592,A -85,B 0,C 180,E1 -3629.34,E2 -3629.34} C_VEL
LIN {X 0,Y 545.044,Z 125.588,A -85,B 0,C 180,E1 -3631.916,E2 -3631.916} C_VEL
LIN {X 0,Y 545.049,Z 125.592,A -85,B 0,C 180,E1 -3634.566,E2 -3634.566} C_VEL
LIN {X 0,Y 545.026,Z 125.592,A -85,B 0,C 180,E1 -3637.305,E2 -3637.305} C_VEL
LIN {X 0,Y 545.057,Z 125.588,A -85,B 0,C 180,E1 -3640.144,E2 -3640.144} C_VEL
LIN {X 0,Y 545.071,Z 125.586,A -85,B 0,C 180,E1 -3643.108,E2 -3643.108} C_VEL
LIN {X 0,Y 545.042,Z 125.593,A -85,B 0,C 180,E1 -3646.227,E2 -3646.227} C_VEL
LIN {X 0,Y 545.075,Z 125.586,A -85,B 0,C 180,E1 -3648.886,E2 -3648.886} C_VEL
LIN {X 0,Y 545.077,Z 125.586,A -85,B 0,C 180,E1 -3650.82,E2 -3650.82} C_VEL
LIN {X 0,Y 545.037,Z 125.59,A -85,B 0,C 180,E1 -3653.621,E2 -3653.621} C_VEL
LIN {X 0,Y 545.062,Z 125.591,A -85,B 0,C 180,E1 -3656.329,E2 -3656.329} C_VEL
LIN {X 0,Y 545.065,Z 125.585,A -85,B 0,C 180,E1 -3658.953,E2 -3658.953} C_VEL
LIN {X 0,Y 545.1,Z 125.584,A -85,B 0,C 180,E1 -3661.509,E2 -3661.509} C_VEL
LIN {X 0,Y 545.094,Z 125.583,A -85,B 0,C 180,E1 -3664.492,E2 -3664.492} C_VEL
LIN {X 0,Y 545.125,Z 125.778,A -85,B 0,C 180,E1 -3665.585,E2 -3665.585} C_VEL
LIN {X 0,Y 546.252,Z 132.956,A -85,B 0,C 180,E1 -3666.696,E2 -3666.696} C_VEL
LIN {X 0,Y 545.934,Z 153.279,A -85,B 0,C 180,E1 -3669.662,E2 -3669.662} C_VEL
LIN {X 0,Y 545.594,Z 174.927,A -85,B 0,C 180,E1 -3672.767,E2 -3672.767} C_VEL
LIN {X 0,Y 545.305,Z 193.74,A -85,B 0,C 180,E1 -3675.436,E2 -3675.436} C_VEL
LIN {X 0,Y 546.524,Z 203.246,A -85,B 0,C 180,E1 -3675.596,E2 -3675.596} C_VEL
LIN {X 0,Y 546.19,Z 302.331,A -85,B 0,C 180,E1 -3676.917,E2 -3676.917} C_VEL
LIN {X 0,Y 546.024,Z 315.618,A -85,B 0,C 180,E1 -3677.244,E2 -3677.244} C_VEL
LIN {X 0,Y 545.84,Z 328.926,A -85,B 0,C 180,E1 -3677.735,E2 -3677.735} C_VEL
LIN {X 0,Y 545.634,Z 340.421,A -85,B 0,C 180,E1 -3678.315,E2 -3678.315} C_VEL
LIN {X 0,Y 545.451,Z 351.725,A -85,B 0,C 180,E1 -3679.045,E2 -3679.045} C_VEL
LIN {X 0,Y 545.231,Z 362.194,A -85,B 0,C 180,E1 -3679.886,E2 -3679.886} C_VEL
LIN {X 0,Y 545.084,Z 370.758,A -85,B 0,C 180,E1 -3680.726,E2 -3680.726} C_VEL
LIN {X 0,Y 544.946,Z 378.662,A -85,B 0,C 180,E1 -3681.658,E2 -3681.658} C_VEL
LIN {X 0,Y 544.823,Z 386.382,A -85,B 0,C 180,E1 -3682.775,E2 -3682.775} C_VEL
LIN {X 0,Y 544.776,Z 393.503,A -85,B 0,C 180,E1 -3684.077,E2 -3684.077} C_VEL
LIN {X 0,Y 544.628,Z 398.235,A -85,B 0,C 180,E1 -3685.189,E2 -3685.189} C_VEL
LIN {X 0,Y 544.669,Z 401.857,A -85,B 0,C 180,E1 -3686.302,E2 -3686.302} C_VEL
LIN {X 0,Y 544.65,Z 403.724,A -85,B 0,C 180,E1 -3687.042,E2 -3687.042} C_VEL
LIN {X 0,Y 544.546,Z 406.118,A -85,B 0,C 180,E1 -3688.522,E2 -3688.522} C_VEL
LIN {X 0,Y 544.542,Z 406.728,A -85,B 0,C 180,E1 -3689.261,E2 -3689.261} C_VEL
LIN {X 0,Y 544.541,Z 406.944,A -85,B 0,C 180,E1 -3690.001,E2 -3690.001} C_VEL
LIN {X 0,Y 544.542,Z 406.727,A -85,B 0,C 180,E1 -3690.74,E2 -3690.74} C_VEL
LIN {X 0,Y 544.572,Z 405.121,A -85,B 0,C 180,E1 -3692.22,E2 -3692.22} C_VEL
LIN {X 0,Y 544.65,Z 403.724,A -85,B 0,C 180,E1 -3692.959,E2 -3692.959} C_VEL
LIN {X 0,Y 544.684,Z 400.78,A -85,B 0,C 180,E1 -3694.07,E2 -3694.07} C_VEL
LIN {X 0,Y 544.654,Z 396.791,A -85,B 0,C 180,E1 -3695.183,E2 -3695.183} C_VEL
LIN {X 0,Y 544.71,Z 391.498,A -85,B 0,C 180,E1 -3696.329,E2 -3696.329} C_VEL
LIN {X 0,Y 544.837,Z 385.205,A -85,B 0,C 180,E1 -3697.412,E2 -3697.412} C_VEL
LIN {X 0,Y 544.972,Z 377.152,A -85,B 0,C 180,E1 -3698.529,E2 -3698.529} C_VEL
LIN {X 0,Y 545.114,Z 368.947,A -85,B 0,C 180,E1 -3699.462,E2 -3699.462} C_VEL
LIN {X 0,Y 545.35,Z 358.947,A -85,B 0,C 180,E1 -3700.395,E2 -3700.395} C_VEL
LIN {X 0,Y 545.531,Z 348.077,A -85,B 0,C 180,E1 -3701.209,E2 -3701.209} C_VEL
LIN {X 0,Y 545.71,Z 336.598,A -85,B 0,C 180,E1 -3701.892,E2 -3701.892} C_VEL
LIN {X 0,Y 545.927,Z 324.35,A -85,B 0,C 180,E1 -3702.453,E2 -3702.453} C_VEL
LIN {X 0,Y 546.112,Z 311.503,A -85,B 0,C 180,E1 -3702.874,E2 -3702.874} C_VEL
LIN {X 0,Y 546.249,Z 297.884,A -85,B 0,C 180,E1 -3703.154,E2 -3703.154} C_VEL
LIN {X 0,Y 546.347,Z 200.874,A -85,B 0,C 180,E1 -3704.44,E2 -3704.44} C_VEL
LIN {X 0,Y 545.321,Z 193.611,A -85,B 0,C 180,E1 -3704.58,E2 -3704.58} C_VEL
LIN {X 0,Y 545.591,Z 173.201,A -85,B 0,C 180,E1 -3707.474,E2 -3707.474} C_VEL
LIN {X 0,Y 545.939,Z 151.86,A -85,B 0,C 180,E1 -3710.536,E2 -3710.536} C_VEL
LIN {X 0,Y 546.211,Z 132.859,A -85,B 0,C 180,E1 -3713.307,E2 -3713.307} C_VEL
LIN {X 0,Y 545.561,Z 127.915,A -85,B 0,C 180,E1 -3714.065,E2 -3714.065} C_VEL
LIN {X 0,Y 545.109,Z 125.586,A -85,B 0,C 180,E1 -3714.468,E2 -3714.468} C_VEL
LIN {X 0,Y 545.06,Z 125.591,A -85,B 0,C 180,E1 -3717.658,E2 -3717.658} C_VEL
LIN {X 0,Y 545.057,Z 125.593,A -85,B 0,C 180,E1 -3720.242,E2 -3720.242} C_VEL
LIN {X 0,Y 545.082,Z 125.584,A -85,B 0,C 180,E1 -3723.062,E2 -3723.062} C_VEL
LIN {X 0,Y 545.027,Z 125.597,A -85,B 0,C 180,E1 -3725.672,E2 -3725.672} C_VEL
LIN {X 0,Y 545.052,Z 125.588,A -85,B 0,C 180,E1 -3728.238,E2 -3728.238} C_VEL
LIN {X 0,Y 545.083,Z 125.582,A -85,B 0,C 180,E1 -3730.473,E2 -3730.473} C_VEL
LIN {X 0,Y 545.046,Z 125.59,A -85,B 0,C 180,E1 -3733.11,E2 -3733.11} C_VEL
LIN {X 0,Y 545.046,Z 125.587,A -85,B 0,C 180,E1 -3736.227,E2 -3736.227} C_VEL
LIN {X 0,Y 545.072,Z 125.587,A -85,B 0,C 180,E1 -3738.884,E2 -3738.884} C_VEL
LIN {X 0,Y 545.047,Z 125.588,A -85,B 0,C 180,E1 -3741.865,E2 -3741.865} C_VEL
LIN {X 0,Y 545.029,Z 125.591,A -85,B 0,C 180,E1 -3744.531,E2 -3744.531} C_VEL
LIN {X 0,Y 545.061,Z 125.592,A -85,B 0,C 180,E1 -3747.211,E2 -3747.211} C_VEL
LIN {X 0,Y 545.062,Z 125.585,A -85,B 0,C 180,E1 -3749.81,E2 -3749.81} C_VEL
LIN {X 0,Y 545.035,Z 125.597,A -85,B 0,C 180,E1 -3752.839,E2 -3752.839} C_VEL
LIN {X 0,Y 545.018,Z 125.59,A -85,B 0,C 180,E1 -3755.629,E2 -3755.629} C_VEL
LIN {X 0,Y 545.062,Z 125.587,A -85,B 0,C 180,E1 -3758.181,E2 -3758.181} C_VEL
LIN {X 0,Y 545.101,Z 125.585,A -85,B 0,C 180,E1 -3760.414,E2 -3760.414} C_VEL
LIN {X 0,Y 545.019,Z 125.59,A -85,B 0,C 180,E1 -3763.519,E2 -3763.519} C_VEL
LIN {X 0,Y 545.06,Z 125.585,A -85,B 0,C 180,E1 -3765.819,E2 -3765.819} C_VEL
LIN {X 0,Y 545.068,Z 125.586,A -85,B 0,C 180,E1 -3768.848,E2 -3768.848} C_VEL
LIN {X 0,Y 545.059,Z 125.587,A -85,B 0,C 180,E1 -3771.846,E2 -3771.846} C_VEL
LIN {X 0,Y 545.155,Z 125.574,A -85,B 0,C 180,E1 -3774.823,E2 -3774.823} C_VEL
LIN {X 0,Y 545.188,Z 125.573,A -85,B 0,C 180,E1 -3777.784,E2 -3777.784} C_VEL
LIN {X 0,Y 545.189,Z 125.577,A -85,B 0,C 180,E1 -3780,E2 -3780} C_VEL
LIN {X 0,Y 545.142,Z 125.572,A -85,B 0,C 180,E1 -3782.956,E2 -3782.956} C_VEL
LIN {X 0,Y 545.125,Z 125.583,A -85,B 0,C 180,E1 -3785.92,E2 -3785.92} C_VEL
LIN {X 0,Y 545.091,Z 125.579,A -85,B 0,C 180,E1 -3788.901,E2 -3788.901} C_VEL
LIN {X 0,Y 545.094,Z 125.584,A -85,B 0,C 180,E1 -3791.905,E2 -3791.905} C_VEL
LIN {X 0,Y 545.076,Z 125.584,A -85,B 0,C 180,E1 -3794.944,E2 -3794.944} C_VEL
LIN {X 0,Y 545.054,Z 125.586,A -85,B 0,C 180,E1 -3798.027,E2 -3798.027} C_VEL
LIN {X 0,Y 545.089,Z 125.58,A -85,B 0,C 180,E1 -3800.372,E2 -3800.372} C_VEL
LIN {X 0,Y 545.07,Z 125.585,A -85,B 0,C 180,E1 -3803.56,E2 -3803.56} C_VEL
LIN {X 0,Y 545.052,Z 125.586,A -85,B 0,C 180,E1 -3806.002,E2 -3806.002} C_VEL
LIN {X 0,Y 545.071,Z 125.59,A -85,B 0,C 180,E1 -3808.745,E2 -3808.745} C_VEL
LIN {X 0,Y 545.059,Z 125.585,A -85,B 0,C 180,E1 -3811.679,E2 -3811.679} C_VEL
LIN {X 0,Y 545.06,Z 125.592,A -85,B 0,C 180,E1 -3814.565,E2 -3814.565} C_VEL
LIN {X 0,Y 545.067,Z 125.588,A -85,B 0,C 180,E1 -3816.964,E2 -3816.964} C_VEL
LIN {X 0,Y 544.354,Z 125.675,A -85,B 0,C 180,E1 -3817.581,E2 -3817.581} C_VEL
LIN {X 0,Y 541.482,Z 126.039,A -85,B 0,C 180,E1 -3818.582,E2 -3818.582} C_VEL
LIN {X 0,Y 539.093,Z 126.331,A -85,B 0,C 180,E1 -3819.387,E2 -3819.387} C_VEL
LIN {X 0,Y 538.085,Z 126.455,A -85,B 0,C 180,E1 -3820.01,E2 -3820.01} C_VEL
LIN {X 0,Y 538.011,Z 126.461,A -85,B 0,C 180,E1 -3820.22,E2 -3820.22} C_VEL
LIN {X 0,Y 538.029,Z 126.463,A -85,B 0,C 180,E1 -3822.988,E2 -3822.988} C_VEL
LIN {X 0,Y 538.006,Z 126.471,A -85,B 0,C 180,E1 -3826.184,E2 -3826.184} C_VEL
LIN {X 0,Y 538.052,Z 126.459,A -85,B 0,C 180,E1 -3829.253,E2 -3829.253} C_VEL
LIN {X 0,Y 537.996,Z 126.474,A -85,B 0,C 180,E1 -3832.122,E2 -3832.122} C_VEL
LIN {X 0,Y 538.002,Z 126.465,A -85,B 0,C 180,E1 -3834.916,E2 -3834.916} C_VEL
LIN {X 0,Y 538.023,Z 126.467,A -85,B 0,C 180,E1 -3837.617,E2 -3837.617} C_VEL
LIN {X 0,Y 538.019,Z 126.467,A -85,B 0,C 180,E1 -3840.239,E2 -3840.239} C_VEL
LIN {X 0,Y 538.055,Z 126.46,A -85,B 0,C 180,E1 -3842.795,E2 -3842.795} C_VEL
LIN {X 0,Y 538.06,Z 126.464,A -85,B 0,C 180,E1 -3845.293,E2 -3845.293} C_VEL
LIN {X 0,Y 538.081,Z 126.552,A -85,B 0,C 180,E1 -3846.256,E2 -3846.256} C_VEL
LIN {X 0,Y 538.418,Z 131.132,A -85,B 0,C 180,E1 -3847.149,E2 -3847.149} C_VEL
LIN {X 0,Y 538.238,Z 147.629,A -85,B 0,C 180,E1 -3850.303,E2 -3850.303} C_VEL
LIN {X 0,Y 539.689,Z 156.408,A -85,B 0,C 180,E1 -3850.469,E2 -3850.469} C_VEL
LIN {X 0,Y 539.311,Z 254.722,A -85,B 0,C 180,E1 -3851.805,E2 -3851.805} C_VEL
LIN {X 0,Y 539.143,Z 268.101,A -85,B 0,C 180,E1 -3852.147,E2 -3852.147} C_VEL
LIN {X 0,Y 538.997,Z 280.002,A -85,B 0,C 180,E1 -3852.597,E2 -3852.597} C_VEL
LIN {X 0,Y 538.82,Z 292.26,A -85,B 0,C 180,E1 -3853.226,E2 -3853.226} C_VEL
LIN {X 0,Y 538.546,Z 303.858,A -85,B 0,C 180,E1 -3853.997,E2 -3853.997} C_VEL
LIN {X 0,Y 538.325,Z 314.26,A -85,B 0,C 180,E1 -3854.864,E2 -3854.864} C_VEL
LIN {X 0,Y 538.144,Z 323.542,A -85,B 0,C 180,E1 -3855.825,E2 -3855.825} C_VEL
LIN {X 0,Y 537.917,Z 332.525,A -85,B 0,C 180,E1 -3856.975,E2 -3856.975} C_VEL
LIN {X 0,Y 537.802,Z 339.717,A -85,B 0,C 180,E1 -3858.122,E2 -3858.122} C_VEL
LIN {X 0,Y 537.665,Z 344.545,A -85,B 0,C 180,E1 -3859.074,E2 -3859.074} C_VEL
LIN {X 0,Y 537.601,Z 349.213,A -85,B 0,C 180,E1 -3860.215,E2 -3860.215} C_VEL
LIN {X 0,Y 537.572,Z 352.757,A -85,B 0,C 180,E1 -3861.352,E2 -3861.352} C_VEL
LIN {X 0,Y 537.546,Z 355.28,A -85,B 0,C 180,E1 -3862.487,E2 -3862.487} C_VEL
LIN {X 0,Y 537.587,Z 356.729,A -85,B 0,C 180,E1 -3863.499,E2 -3863.499} C_VEL
LIN {X 0,Y 537.524,Z 357.534,A -85,B 0,C 180,E1 -3864.748,E2 -3864.748} C_VEL
LIN {X 0,Y 537.562,Z 357.079,A -85,B 0,C 180,E1 -3866.251,E2 -3866.251} C_VEL
LIN {X 0,Y 537.575,Z 356.229,A -85,B 0,C 180,E1 -3867.002,E2 -3867.002} C_VEL
LIN {X 0,Y 537.476,Z 353.359,A -85,B 0,C 180,E1 -3868.501,E2 -3868.501} C_VEL
LIN {X 0,Y 537.586,Z 350.07,A -85,B 0,C 180,E1 -3869.625,E2 -3869.625} C_VEL
LIN {X 0,Y 537.577,Z 345.74,A -85,B 0,C 180,E1 -3870.748,E2 -3870.748} C_VEL
LIN {X 0,Y 537.794,Z 340.224,A -85,B 0,C 180,E1 -3871.872,E2 -3871.872} C_VEL
LIN {X 0,Y 537.792,Z 333.377,A -85,B 0,C 180,E1 -3872.996,E2 -3872.996} C_VEL
LIN {X 0,Y 538.1,Z 324.78,A -85,B 0,C 180,E1 -3874.119,E2 -3874.119} C_VEL
LIN {X 0,Y 538.247,Z 316.014,A -85,B 0,C 180,E1 -3875.056,E2 -3875.056} C_VEL
LIN {X 0,Y 538.496,Z 306.382,A -85,B 0,C 180,E1 -3875.898,E2 -3875.898} C_VEL
LIN {X 0,Y 538.727,Z 295.826,A -85,B 0,C 180,E1 -3876.648,E2 -3876.648} C_VEL
LIN {X 0,Y 538.962,Z 284.427,A -85,B 0,C 180,E1 -3877.284,E2 -3877.284} C_VEL
LIN {X 0,Y 539.104,Z 271.501,A -85,B 0,C 180,E1 -3877.829,E2 -3877.829} C_VEL
LIN {X 0,Y 539.287,Z 259.249,A -85,B 0,C 180,E1 -3878.189,E2 -3878.189} C_VEL
LIN {X 0,Y 539.339,Z 245.62,A -85,B 0,C 180,E1 -3878.429,E2 -3878.429} C_VEL
LIN {X 0,Y 539.654,Z 155.292,A -85,B 0,C 180,E1 -3879.636,E2 -3879.636} C_VEL
LIN {X 0,Y 538.196,Z 147.597,A -85,B 0,C 180,E1 -3879.797,E2 -3879.797} C_VEL
LIN {X 0,Y 538.363,Z 132.778,A -85,B 0,C 180,E1 -3882.63,E2 -3882.63} C_VEL
LIN {X 0,Y 538.134,Z 126.813,A -85,B 0,C 180,E1 -3883.788,E2 -3883.788} C_VEL
LIN {X 0,Y 538.054,Z 126.465,A -85,B 0,C 180,E1 -3883.886,E2 -3883.886} C_VEL
LIN {X 0,Y 538.014,Z 126.469,A -85,B 0,C 180,E1 -3886.7,E2 -3886.7} C_VEL
LIN {X 0,Y 538.085,Z 126.457,A -85,B 0,C 180,E1 -3889.88,E2 -3889.88} C_VEL
LIN {X 0,Y 538.014,Z 126.463,A -85,B 0,C 180,E1 -3893.071,E2 -3893.071} C_VEL
LIN {X 0,Y 538.043,Z 126.463,A -85,B 0,C 180,E1 -3895.671,E2 -3895.671} C_VEL
LIN {X 0,Y 538.025,Z 126.471,A -85,B 0,C 180,E1 -3898.05,E2 -3898.05} C_VEL
LIN {X 0,Y 538.019,Z 126.464,A -85,B 0,C 180,E1 -3900.626,E2 -3900.626} C_VEL
LIN {X 0,Y 538.043,Z 126.462,A -85,B 0,C 180,E1 -3903.282,E2 -3903.282} C_VEL
LIN {X 0,Y 537.991,Z 126.472,A -85,B 0,C 180,E1 -3906.003,E2 -3906.003} C_VEL
LIN {X 0,Y 538.01,Z 126.464,A -85,B 0,C 180,E1 -3908.829,E2 -3908.829} C_VEL
LIN {X 0,Y 538.025,Z 126.468,A -85,B 0,C 180,E1 -3911.772,E2 -3911.772} C_VEL
LIN {X 0,Y 538,Z 126.467,A -85,B 0,C 180,E1 -3914.861,E2 -3914.861} C_VEL
LIN {X 0,Y 538.012,Z 126.47,A -85,B 0,C 180,E1 -3917.213,E2 -3917.213} C_VEL
LIN {X 0,Y 538.013,Z 126.464,A -85,B 0,C 180,E1 -3920.202,E2 -3920.202} C_VEL
LIN {X 0,Y 538.015,Z 126.469,A -85,B 0,C 180,E1 -3923.066,E2 -3923.066} C_VEL
LIN {X 0,Y 538.001,Z 126.466,A -85,B 0,C 180,E1 -3925.825,E2 -3925.825} C_VEL
LIN {X 0,Y 537.998,Z 126.468,A -85,B 0,C 180,E1 -3928.498,E2 -3928.498} C_VEL
LIN {X 0,Y 538.009,Z 126.471,A -85,B 0,C 180,E1 -3931.097,E2 -3931.097} C_VEL
LIN {X 0,Y 538.014,Z 126.465,A -85,B 0,C 180,E1 -3933.632,E2 -3933.632} C_VEL
LIN {X 0,Y 537.995,Z 126.473,A -85,B 0,C 180,E1 -3936.927,E2 -3936.927} C_VEL
LIN {X 0,Y 538.069,Z 126.46,A -85,B 0,C 180,E1 -3940.147,E2 -3940.147} C_VEL
LIN {X 0,Y 537.972,Z 126.47,A -85,B 0,C 180,E1 -3943.297,E2 -3943.297} C_VEL
LIN {X 0,Y 538.029,Z 126.463,A -85,B 0,C 180,E1 -3945.63,E2 -3945.63} C_VEL
LIN {X 0,Y 538.063,Z 126.462,A -85,B 0,C 180,E1 -3948.701,E2 -3948.701} C_VEL
LIN {X 0,Y 538.042,Z 126.463,A -85,B 0,C 180,E1 -3951.739,E2 -3951.739} C_VEL
LIN {X 0,Y 538.113,Z 126.454,A -85,B 0,C 180,E1 -3954.754,E2 -3954.754} C_VEL
LIN {X 0,Y 538.151,Z 126.452,A -85,B 0,C 180,E1 -3957.755,E2 -3957.755} C_VEL
LIN {X 0,Y 538.147,Z 126.454,A -85,B 0,C 180,E1 -3960,E2 -3960} C_VEL
LIN {X 0,Y 538.1,Z 126.454,A -85,B 0,C 180,E1 -3962.995,E2 -3962.995} C_VEL
LIN {X 0,Y 538.096,Z 126.46,A -85,B 0,C 180,E1 -3965.998,E2 -3965.998} C_VEL
LIN {X 0,Y 538.034,Z 126.463,A -85,B 0,C 180,E1 -3969.018,E2 -3969.018} C_VEL
LIN {X 0,Y 538.045,Z 126.463,A -85,B 0,C 180,E1 -3972.063,E2 -3972.063} C_VEL
LIN {X 0,Y 538.025,Z 126.467,A -85,B 0,C 180,E1 -3975.144,E2 -3975.144} C_VEL
LIN {X 0,Y 537.996,Z 126.466,A -85,B 0,C 180,E1 -3978.271,E2 -3978.271} C_VEL
LIN {X 0,Y 538.023,Z 126.464,A -85,B 0,C 180,E1 -3980.652,E2 -3980.652} C_VEL
LIN {X 0,Y 537.994,Z 126.468,A -85,B 0,C 180,E1 -3983.878,E2 -3983.878} C_VEL
LIN {X 0,Y 538.023,Z 126.463,A -85,B 0,C 180,E1 -3986.368,E2 -3986.368} C_VEL
LIN {X 0,Y 538.019,Z 126.471,A -85,B 0,C 180,E1 -3988.934,E2 -3988.934} C_VEL
LIN {X 0,Y 537.999,Z 126.466,A -85,B 0,C 180,E1 -3991.888,E2 -3991.888} C_VEL
LIN {X 0,Y 537.999,Z 126.471,A -85,B 0,C 180,E1 -3994.618,E2 -3994.618} C_VEL
LIN {X 0,Y 537.995,Z 126.47,A -85,B 0,C 180,E1 -3997.171,E2 -3997.171} C_VEL
LIN {X 0,Y 538.013,Z 126.464,A -85,B 0,C 180,E1 -3999.798,E2 -3999.798} C_VEL
LIN {X 0,Y 538.011,Z 126.469,A -85,B 0,C 180,E1 -4002.787,E2 -4002.787} C_VEL
LIN {X 0,Y 538.012,Z 126.466,A -85,B 0,C 180,E1 -4005.928,E2 -4005.928} C_VEL
LIN {X 0,Y 538.024,Z 126.469,A -85,B 0,C 180,E1 -4008.228,E2 -4008.228} C_VEL
LIN {X 0,Y 538.009,Z 126.464,A -85,B 0,C 180,E1 -4011.171,E2 -4011.171} C_VEL
LIN {X 0,Y 537.989,Z 126.473,A -85,B 0,C 180,E1 -4014.09,E2 -4014.09} C_VEL
LIN {X 0,Y 538.026,Z 126.463,A -85,B 0,C 180,E1 -4016.728,E2 -4016.728} C_VEL
LIN {X 0,Y 538.024,Z 126.464,A -85,B 0,C 180,E1 -4019.557,E2 -4019.557} C_VEL
LIN {X 0,Y 538.055,Z 126.459,A -85,B 0,C 180,E1 -4022.649,E2 -4022.649} C_VEL
LIN {X 0,Y 538.072,Z 126.559,A -85,B 0,C 180,E1 -4025.412,E2 -4025.412} C_VEL
LIN {X 0,Y 539.304,Z 134.003,A -85,B 0,C 180,E1 -4026.581,E2 -4026.581} C_VEL
LIN {X 0,Y 538.992,Z 151.611,A -85,B 0,C 180,E1 -4029.188,E2 -4029.188} C_VEL
LIN {X 0,Y 538.585,Z 172.864,A -85,B 0,C 180,E1 -4032.285,E2 -4032.285} C_VEL
LIN {X 0,Y 538.305,Z 190.784,A -85,B 0,C 180,E1 -4034.865,E2 -4034.865} C_VEL
LIN {X 0,Y 538.264,Z 193.37,A -85,B 0,C 180,E1 -4035.235,E2 -4035.235} C_VEL
LIN {X 0,Y 539.629,Z 203.321,A -85,B 0,C 180,E1 -4035.413,E2 -4035.413} C_VEL
LIN {X 0,Y 539.293,Z 302.003,A -85,B 0,C 180,E1 -4036.746,E2 -4036.746} C_VEL
LIN {X 0,Y 539.107,Z 315.292,A -85,B 0,C 180,E1 -4037.077,E2 -4037.077} C_VEL
LIN {X 0,Y 538.899,Z 327.476,A -85,B 0,C 180,E1 -4037.527,E2 -4037.527} C_VEL
LIN {X 0,Y 538.679,Z 339.434,A -85,B 0,C 180,E1 -4038.123,E2 -4038.123} C_VEL
LIN {X 0,Y 538.456,Z 351.4,A -85,B 0,C 180,E1 -4038.901,E2 -4038.901} C_VEL
LIN {X 0,Y 538.192,Z 361.869,A -85,B 0,C 180,E1 -4039.752,E2 -4039.752} C_VEL
LIN {X 0,Y 538.046,Z 370.434,A -85,B 0,C 180,E1 -4040.604,E2 -4040.604} C_VEL
LIN {X 0,Y 537.891,Z 378.337,A -85,B 0,C 180,E1 -4041.548,E2 -4041.548} C_VEL
LIN {X 0,Y 537.754,Z 386.059,A -85,B 0,C 180,E1 -4042.68,E2 -4042.68} C_VEL
LIN {X 0,Y 537.665,Z 393.178,A -85,B 0,C 180,E1 -4043.998,E2 -4043.998} C_VEL
LIN {X 0,Y 537.54,Z 397.912,A -85,B 0,C 180,E1 -4045.126,E2 -4045.126} C_VEL
LIN {X 0,Y 537.591,Z 401.535,A -85,B 0,C 180,E1 -4046.253,E2 -4046.253} C_VEL
LIN {X 0,Y 537.58,Z 403.401,A -85,B 0,C 180,E1 -4047.003,E2 -4047.003} C_VEL
LIN {X 0,Y 537.452,Z 405.795,A -85,B 0,C 180,E1 -4048.502,E2 -4048.502} C_VEL
LIN {X 0,Y 537.449,Z 406.404,A -85,B 0,C 180,E1 -4049.251,E2 -4049.251} C_VEL
LIN {X 0,Y 537.449,Z 406.621,A -85,B 0,C 180,E1 -4050.001,E2 -4050.001} C_VEL
LIN {X 0,Y 537.449,Z 406.404,A -85,B 0,C 180,E1 -4050.75,E2 -4050.75} C_VEL
LIN {X 0,Y 537.49,Z 404.797,A -85,B 0,C 180,E1 -4052.249,E2 -4052.249} C_VEL
LIN {X 0,Y 537.58,Z 403.4,A -85,B 0,C 180,E1 -4052.998,E2 -4052.998} C_VEL
LIN {X 0,Y 537.603,Z 400.454,A -85,B 0,C 180,E1 -4054.124,E2 -4054.124} C_VEL
LIN {X 0,Y 537.588,Z 396.465,A -85,B 0,C 180,E1 -4055.251,E2 -4055.251} C_VEL
LIN {X 0,Y 537.645,Z 390.403,A -85,B 0,C 180,E1 -4056.555,E2 -4056.555} C_VEL
LIN {X 0,Y 537.784,Z 383.636,A -85,B 0,C 180,E1 -4057.699,E2 -4057.699} C_VEL
LIN {X 0,Y 537.931,Z 375.326,A -85,B 0,C 180,E1 -4058.831,E2 -4058.831} C_VEL
LIN {X 0,Y 538.091,Z 366.81,A -85,B 0,C 180,E1 -4059.776,E2 -4059.776} C_VEL
LIN {X 0,Y 538.351,Z 356.294,A -85,B 0,C 180,E1 -4060.722,E2 -4060.722} C_VEL
LIN {X 0,Y 538.583,Z 345.093,A -85,B 0,C 180,E1 -4061.532,E2 -4061.532} C_VEL
LIN {X 0,Y 538.796,Z 334.494,A -85,B 0,C 180,E1 -4062.142,E2 -4062.142} C_VEL
LIN {X 0,Y 539,Z 322.802,A -85,B 0,C 180,E1 -4062.664,E2 -4062.664} C_VEL
LIN {X 0,Y 539.171,Z 309.334,A -85,B 0,C 180,E1 -4063.09,E2 -4063.09} C_VEL
LIN {X 0,Y 539.369,Z 296.025,A -85,B 0,C 180,E1 -4063.349,E2 -4063.349} C_VEL
LIN {X 0,Y 539.508,Z 201.907,A -85,B 0,C 180,E1 -4064.609,E2 -4064.609} C_VEL
LIN {X 0,Y 538.253,Z 193.216,A -85,B 0,C 180,E1 -4064.784,E2 -4064.784} C_VEL
LIN {X 0,Y 538.582,Z 174.546,A -85,B 0,C 180,E1 -4067.466,E2 -4067.466} C_VEL
LIN {X 0,Y 538.955,Z 152.888,A -85,B 0,C 180,E1 -4070.615,E2 -4070.615} C_VEL
LIN {X 0,Y 539.307,Z 135.262,A -85,B 0,C 180,E1 -4073.217,E2 -4073.217} C_VEL
LIN {X 0,Y 538.733,Z 129.86,A -85,B 0,C 180,E1 -4074.051,E2 -4074.051} C_VEL
LIN {X 0,Y 538.064,Z 126.463,A -85,B 0,C 180,E1 -4074.614,E2 -4074.614} C_VEL
LIN {X 0,Y 538.033,Z 126.464,A -85,B 0,C 180,E1 -4077.346,E2 -4077.346} C_VEL
LIN {X 0,Y 538.014,Z 126.472,A -85,B 0,C 180,E1 -4079.762,E2 -4079.762} C_VEL
LIN {X 0,Y 538.021,Z 126.466,A -85,B 0,C 180,E1 -4082.383,E2 -4082.383} C_VEL
LIN {X 0,Y 537.997,Z 126.466,A -85,B 0,C 180,E1 -4085.085,E2 -4085.085} C_VEL
LIN {X 0,Y 537.991,Z 126.472,A -85,B 0,C 180,E1 -4087.878,E2 -4087.878} C_VEL
LIN {X 0,Y 538.049,Z 126.459,A -85,B 0,C 180,E1 -4090.776,E2 -4090.776} C_VEL
LIN {X 0,Y 538.019,Z 126.464,A -85,B 0,C 180,E1 -4094.073,E2 -4094.073} C_VEL
LIN {X 0,Y 537.981,Z 126.471,A -85,B 0,C 180,E1 -4097.018,E2 -4097.018} C_VEL
LIN {X 0,Y 538.023,Z 126.47,A -85,B 0,C 180,E1 -4099.256,E2 -4099.256} C_VEL
LIN {X 0,Y 537.989,Z 126.466,A -85,B 0,C 180,E1 -4102.122,E2 -4102.122} C_VEL
LIN {X 0,Y 537.993,Z 126.472,A -85,B 0,C 180,E1 -4104.915,E2 -4104.915} C_VEL
LIN {X 0,Y 538.011,Z 126.465,A -85,B 0,C 180,E1 -4107.617,E2 -4107.617} C_VEL
LIN {X 0,Y 537.997,Z 126.466,A -85,B 0,C 180,E1 -4110.238,E2 -4110.238} C_VEL
LIN {X 0,Y 538.008,Z 126.472,A -85,B 0,C 180,E1 -4112.793,E2 -4112.793} C_VEL
LIN {X 0,Y 537.98,Z 126.469,A -85,B 0,C 180,E1 -4115.289,E2 -4115.289} C_VEL
LIN {X 0,Y 538.009,Z 126.465,A -85,B 0,C 180,E1 -4118.044,E2 -4118.044} C_VEL
LIN {X 0,Y 538.003,Z 126.467,A -85,B 0,C 180,E1 -4120.939,E2 -4120.939} C_VEL
LIN {X 0,Y 537.967,Z 126.469,A -85,B 0,C 180,E1 -4123.297,E2 -4123.297} C_VEL
LIN {X 0,Y 538.034,Z 126.458,A -85,B 0,C 180,E1 -4125.63,E2 -4125.63} C_VEL
LIN {X 0,Y 538.021,Z 126.465,A -85,B 0,C 180,E1 -4128.7,E2 -4128.7} C_VEL
LIN {X 0,Y 538.028,Z 126.461,A -85,B 0,C 180,E1 -4131.739,E2 -4131.739} C_VEL
LIN {X 0,Y 538.115,Z 126.451,A -85,B 0,C 180,E1 -4134.755,E2 -4134.755} C_VEL
LIN {X 0,Y 538.159,Z 126.448,A -85,B 0,C 180,E1 -4137.755,E2 -4137.755} C_VEL
LIN {X 0,Y 538.157,Z 126.453,A -85,B 0,C 180,E1 -4140,E2 -4140} C_VEL
LIN {X 0,Y 538.11,Z 126.448,A -85,B 0,C 180,E1 -4142.995,E2 -4142.995} C_VEL
LIN {X 0,Y 538.08,Z 126.459,A -85,B 0,C 180,E1 -4145.998,E2 -4145.998} C_VEL
LIN {X 0,Y 538.044,Z 126.458,A -85,B 0,C 180,E1 -4149.018,E2 -4149.018} C_VEL
LIN {X 0,Y 538.053,Z 126.459,A -85,B 0,C 180,E1 -4152.063,E2 -4152.063} C_VEL
LIN {X 0,Y 538.037,Z 126.463,A -85,B 0,C 180,E1 -4155.144,E2 -4155.144} C_VEL
LIN {X 0,Y 538.008,Z 126.463,A -85,B 0,C 180,E1 -4158.271,E2 -4158.271} C_VEL
LIN {X 0,Y 538.035,Z 126.461,A -85,B 0,C 180,E1 -4160.652,E2 -4160.652} C_VEL
LIN {X 0,Y 538.006,Z 126.462,A -85,B 0,C 180,E1 -4163.878,E2 -4163.878} C_VEL
LIN {X 0,Y 538.025,Z 126.463,A -85,B 0,C 180,E1 -4166.368,E2 -4166.368} C_VEL
LIN {X 0,Y 538.031,Z 126.468,A -85,B 0,C 180,E1 -4168.933,E2 -4168.933} C_VEL
LIN {X 0,Y 538.01,Z 126.463,A -85,B 0,C 180,E1 -4171.887,E2 -4171.887} C_VEL
LIN {X 0,Y 538.01,Z 126.471,A -85,B 0,C 180,E1 -4174.617,E2 -4174.617} C_VEL
LIN {X 0,Y 538.005,Z 126.466,A -85,B 0,C 180,E1 -4177.17,E2 -4177.17} C_VEL
LIN {X 0,Y 538.011,Z 126.461,A -85,B 0,C 180,E1 -4180.22,E2 -4180.22} C_VEL
LIN {X 0,Y 537.366,Z 126.544,A -85,B 0,C 180,E1 -4180.845,E2 -4180.845} C_VEL
LIN {X 0,Y 534.52,Z 126.898,A -85,B 0,C 180,E1 -4181.86,E2 -4181.86} C_VEL
LIN {X 0,Y 532.096,Z 127.206,A -85,B 0,C 180,E1 -4182.678,E2 -4182.678} C_VEL
LIN {X 0,Y 531.045,Z 127.332,A -85,B 0,C 180,E1 -4183.309,E2 -4183.309} C_VEL
LIN {X 0,Y 530.956,Z 127.342,A -85,B 0,C 180,E1 -4183.522,E2 -4183.522} C_VEL
LIN {X 0,Y 530.947,Z 127.349,A -85,B 0,C 180,E1 -4186.503,E2 -4186.503} C_VEL
LIN {X 0,Y 530.985,Z 127.34,A -85,B 0,C 180,E1 -4189.567,E2 -4189.567} C_VEL
LIN {X 0,Y 530.971,Z 127.343,A -85,B 0,C 180,E1 -4192.577,E2 -4192.577} C_VEL
LIN {X 0,Y 530.986,Z 127.34,A -85,B 0,C 180,E1 -4195.31,E2 -4195.31} C_VEL
LIN {X 0,Y 530.971,Z 127.347,A -85,B 0,C 180,E1 -4198.032,E2 -4198.032} C_VEL
LIN {X 0,Y 530.993,Z 127.339,A -85,B 0,C 180,E1 -4200.874,E2 -4200.874} C_VEL
LIN {X 0,Y 531.002,Z 127.342,A -85,B 0,C 180,E1 -4203.256,E2 -4203.256} C_VEL
LIN {X 0,Y 531.037,Z 127.468,A -85,B 0,C 180,E1 -4206.161,E2 -4206.161} C_VEL
LIN {X 0,Y 531.436,Z 131.918,A -85,B 0,C 180,E1 -4207.037,E2 -4207.037} C_VEL
LIN {X 0,Y 531.251,Z 147.883,A -85,B 0,C 180,E1 -4210.103,E2 -4210.103} C_VEL
LIN {X 0,Y 532.807,Z 156.46,A -85,B 0,C 180,E1 -4210.273,E2 -4210.273} C_VEL
LIN {X 0,Y 532.426,Z 254.55,A -85,B 0,C 180,E1 -4211.62,E2 -4211.62} C_VEL
LIN {X 0,Y 532.239,Z 268.37,A -85,B 0,C 180,E1 -4211.975,E2 -4211.975} C_VEL
LIN {X 0,Y 532.072,Z 281.007,A -85,B 0,C 180,E1 -4212.462,E2 -4212.462} C_VEL
LIN {X 0,Y 531.863,Z 293.068,A -85,B 0,C 180,E1 -4213.099,E2 -4213.099} C_VEL
LIN {X 0,Y 531.604,Z 303.269,A -85,B 0,C 180,E1 -4213.782,E2 -4213.782} C_VEL
LIN {X 0,Y 531.333,Z 313.836,A -85,B 0,C 180,E1 -4214.66,E2 -4214.66} C_VEL
LIN {X 0,Y 531.145,Z 323.294,A -85,B 0,C 180,E1 -4215.635,E2 -4215.635} C_VEL
LIN {X 0,Y 530.878,Z 332.374,A -85,B 0,C 180,E1 -4216.799,E2 -4216.799} C_VEL
LIN {X 0,Y 530.749,Z 339.659,A -85,B 0,C 180,E1 -4217.962,E2 -4217.962} C_VEL
LIN {X 0,Y 530.621,Z 344.553,A -85,B 0,C 180,E1 -4218.927,E2 -4218.927} C_VEL
LIN {X 0,Y 530.549,Z 349.289,A -85,B 0,C 180,E1 -4220.083,E2 -4220.083} C_VEL
LIN {X 0,Y 530.494,Z 352.896,A -85,B 0,C 180,E1 -4221.236,E2 -4221.236} C_VEL
LIN {X 0,Y 530.455,Z 355.479,A -85,B 0,C 180,E1 -4222.386,E2 -4222.386} C_VEL
LIN {X 0,Y 530.518,Z 357.07,A -85,B 0,C 180,E1 -4223.496,E2 -4223.496} C_VEL
LIN {X 0,Y 530.45,Z 357.843,A -85,B 0,C 180,E1 -4224.678,E2 -4224.678} C_VEL
LIN {X 0,Y 530.481,Z 357.448,A -85,B 0,C 180,E1 -4226.201,E2 -4226.201} C_VEL
LIN {X 0,Y 530.506,Z 356.648,A -85,B 0,C 180,E1 -4226.962,E2 -4226.962} C_VEL
LIN {X 0,Y 530.388,Z 353.836,A -85,B 0,C 180,E1 -4228.481,E2 -4228.481} C_VEL
LIN {X 0,Y 530.499,Z 350.606,A -85,B 0,C 180,E1 -4229.62,E2 -4229.62} C_VEL
LIN {X 0,Y 530.504,Z 346.34,A -85,B 0,C 180,E1 -4230.758,E2 -4230.758} C_VEL
LIN {X 0,Y 530.716,Z 340.894,A -85,B 0,C 180,E1 -4231.896,E2 -4231.896} C_VEL
LIN {X 0,Y 530.743,Z 334.133,A -85,B 0,C 180,E1 -4233.035,E2 -4233.035} C_VEL
LIN {X 0,Y 531.067,Z 325.66,A -85,B 0,C 180,E1 -4234.173,E2 -4234.173} C_VEL
LIN {X 0,Y 531.234,Z 317.004,A -85,B 0,C 180,E1 -4235.123,E2 -4235.123} C_VEL
LIN {X 0,Y 531.527,Z 306.352,A -85,B 0,C 180,E1 -4236.071,E2 -4236.071} C_VEL
LIN {X 0,Y 531.798,Z 295.679,A -85,B 0,C 180,E1 -4236.83,E2 -4236.83} C_VEL
LIN {X 0,Y 532.071,Z 283.55,A -85,B 0,C 180,E1 -4237.503,E2 -4237.503} C_VEL
LIN {X 0,Y 532.238,Z 270.773,A -85,B 0,C 180,E1 -4238.036,E2 -4238.036} C_VEL
LIN {X 0,Y 532.385,Z 258.031,A -85,B 0,C 180,E1 -4238.396,E2 -4238.396} C_VEL
LIN {X 0,Y 532.473,Z 242.02,A -85,B 0,C 180,E1 -4238.658,E2 -4238.658} C_VEL
LIN {X 0,Y 532.867,Z 156.676,A -85,B 0,C 180,E1 -4239.812,E2 -4239.812} C_VEL
LIN {X 0,Y 531.195,Z 147.813,A -85,B 0,C 180,E1 -4239.999,E2 -4239.999} C_VEL
LIN {X 0,Y 531.414,Z 132.257,A -85,B 0,C 180,E1 -4242.992,E2 -4242.992} C_VEL
LIN {X 0,Y 531.01,Z 127.343,A -85,B 0,C 180,E1 -4243.977,E2 -4243.977} C_VEL
LIN {X 0,Y 530.972,Z 127.344,A -85,B 0,C 180,E1 -4246.928,E2 -4246.928} C_VEL
LIN {X 0,Y 531.026,Z 127.341,A -85,B 0,C 180,E1 -4250.126,E2 -4250.126} C_VEL
LIN {X 0,Y 530.945,Z 127.347,A -85,B 0,C 180,E1 -4252.572,E2 -4252.572} C_VEL
LIN {X 0,Y 530.994,Z 127.338,A -85,B 0,C 180,E1 -4255.057,E2 -4255.057} C_VEL
LIN {X 0,Y 531.008,Z 127.339,A -85,B 0,C 180,E1 -4257.595,E2 -4257.595} C_VEL
LIN {X 0,Y 530.972,Z 127.341,A -85,B 0,C 180,E1 -4260.644,E2 -4260.644} C_VEL
LIN {X 0,Y 530.984,Z 127.346,A -85,B 0,C 180,E1 -4263.772,E2 -4263.772} C_VEL
LIN {X 0,Y 530.951,Z 127.344,A -85,B 0,C 180,E1 -4266.557,E2 -4266.557} C_VEL
LIN {X 0,Y 530.984,Z 127.345,A -85,B 0,C 180,E1 -4269.442,E2 -4269.442} C_VEL
LIN {X 0,Y 530.972,Z 127.341,A -85,B 0,C 180,E1 -4272.456,E2 -4272.456} C_VEL
LIN {X 0,Y 530.97,Z 127.348,A -85,B 0,C 180,E1 -4275.621,E2 -4275.621} C_VEL
LIN {X 0,Y 530.986,Z 127.34,A -85,B 0,C 180,E1 -4278.563,E2 -4278.563} C_VEL
LIN {X 0,Y 530.947,Z 127.349,A -85,B 0,C 180,E1 -4281.528,E2 -4281.528} C_VEL
LIN {X 0,Y 530.945,Z 127.345,A -85,B 0,C 180,E1 -4284.379,E2 -4284.379} C_VEL
LIN {X 0,Y 530.957,Z 127.35,A -85,B 0,C 180,E1 -4287.132,E2 -4287.132} C_VEL
LIN {X 0,Y 530.95,Z 127.345,A -85,B 0,C 180,E1 -4289.802,E2 -4289.802} C_VEL
LIN {X 0,Y 530.998,Z 127.342,A -85,B 0,C 180,E1 -4292.468,E2 -4292.468} C_VEL
LIN {X 0,Y 530.939,Z 127.352,A -85,B 0,C 180,E1 -4294.939,E2 -4294.939} C_VEL
LIN {X 0,Y 530.964,Z 127.343,A -85,B 0,C 180,E1 -4297.898,E2 -4297.898} C_VEL
LIN {X 0,Y 530.969,Z 127.348,A -85,B 0,C 180,E1 -4300.676,E2 -4300.676} C_VEL
LIN {X 0,Y 530.94,Z 127.348,A -85,B 0,C 180,E1 -4303.069,E2 -4303.069} C_VEL
LIN {X 0,Y 530.989,Z 127.34,A -85,B 0,C 180,E1 -4305.435,E2 -4305.435} C_VEL
LIN {X 0,Y 531.021,Z 127.342,A -85,B 0,C 180,E1 -4308.549,E2 -4308.549} C_VEL
LIN {X 0,Y 531.018,Z 127.337,A -85,B 0,C 180,E1 -4311.629,E2 -4311.629} C_VEL
LIN {X 0,Y 531.074,Z 127.331,A -85,B 0,C 180,E1 -4314.685,E2 -4314.685} C_VEL
LIN {X 0,Y 531.122,Z 127.327,A -85,B 0,C 180,E1 -4317.725,E2 -4317.725} C_VEL
LIN {X 0,Y 531.115,Z 127.329,A -85,B 0,C 180,E1 -4320,E2 -4320} C_VEL
LIN {X 0,Y 531.122,Z 127.327,A -85,B 0,C 180,E1 -4322.275,E2 -4322.275} C_VEL
LIN {X 0,Y 531.079,Z 127.331,A -85,B 0,C 180,E1 -4325.315,E2 -4325.315} C_VEL
LIN {X 0,Y 531.018,Z 127.337,A -85,B 0,C 180,E1 -4328.371,E2 -4328.371} C_VEL
LIN {X 0,Y 531.036,Z 127.339,A -85,B 0,C 180,E1 -4331.671,E2 -4331.671} C_VEL
LIN {X 0,Y 531.007,Z 127.339,A -85,B 0,C 180,E1 -4334.951,E2 -4334.951} C_VEL
LIN {X 0,Y 530.967,Z 127.347,A -85,B 0,C 180,E1 -4337.724,E2 -4337.724} C_VEL
LIN {X 0,Y 531.012,Z 127.337,A -85,B 0,C 180,E1 -4340.128,E2 -4340.128} C_VEL
LIN {X 0,Y 530.929,Z 127.348,A -85,B 0,C 180,E1 -4342.574,E2 -4342.574} C_VEL
LIN {X 0,Y 530.944,Z 127.352,A -85,B 0,C 180,E1 -4345.061,E2 -4345.061} C_VEL
LIN {X 0,Y 530.999,Z 127.34,A -85,B 0,C 180,E1 -4347.596,E2 -4347.596} C_VEL
LIN {X 0,Y 530.956,Z 127.347,A -85,B 0,C 180,E1 -4350.644,E2 -4350.644} C_VEL
LIN {X 0,Y 530.952,Z 127.345,A -85,B 0,C 180,E1 -4353.5,E2 -4353.5} C_VEL
LIN {X 0,Y 530.936,Z 127.347,A -85,B 0,C 180,E1 -4356.154,E2 -4356.154} C_VEL
LIN {X 0,Y 530.957,Z 127.351,A -85,B 0,C 180,E1 -4358.654,E2 -4358.654} C_VEL
LIN {X 0,Y 530.985,Z 127.34,A -85,B 0,C 180,E1 -4361.437,E2 -4361.437} C_VEL
LIN {X 0,Y 530.967,Z 127.348,A -85,B 0,C 180,E1 -4364.549,E2 -4364.549} C_VEL
LIN {X 0,Y 530.975,Z 127.342,A -85,B 0,C 180,E1 -4367.835,E2 -4367.835} C_VEL
LIN {X 0,Y 530.983,Z 127.344,A -85,B 0,C 180,E1 -4370.558,E2 -4370.558} C_VEL
LIN {X 0,Y 530.95,Z 127.344,A -85,B 0,C 180,E1 -4373.443,E2 -4373.443} C_VEL
LIN {X 0,Y 530.995,Z 127.341,A -85,B 0,C 180,E1 -4376.495,E2 -4376.495} C_VEL
LIN {X 0,Y 530.971,Z 127.341,A -85,B 0,C 180,E1 -4379.356,E2 -4379.356} C_VEL
LIN {X 0,Y 531.013,Z 127.338,A -85,B 0,C 180,E1 -4382.468,E2 -4382.468} C_VEL
LIN {X 0,Y 531.06,Z 127.469,A -85,B 0,C 180,E1 -4385.26,E2 -4385.26} C_VEL
LIN {X 0,Y 532.355,Z 135.03,A -85,B 0,C 180,E1 -4386.463,E2 -4386.463} C_VEL
LIN {X 0,Y 532.021,Z 152.653,A -85,B 0,C 180,E1 -4389.105,E2 -4389.105} C_VEL
LIN {X 0,Y 531.591,Z 174.277,A -85,B 0,C 180,E1 -4392.298,E2 -4392.298} C_VEL
LIN {X 0,Y 531.26,Z 193.181,A -85,B 0,C 180,E1 -4395.044,E2 -4395.044} C_VEL
LIN {X 0,Y 532.753,Z 204.281,A -85,B 0,C 180,E1 -4395.238,E2 -4395.238} C_VEL
LIN {X 0,Y 532.387,Z 301.674,A -85,B 0,C 180,E1 -4396.571,E2 -4396.571} C_VEL
LIN {X 0,Y 532.221,Z 314.203,A -85,B 0,C 180,E1 -4396.883,E2 -4396.883} C_VEL
LIN {X 0,Y 531.951,Z 327.15,A -85,B 0,C 180,E1 -4397.361,E2 -4397.361} C_VEL
LIN {X 0,Y 531.709,Z 339.552,A -85,B 0,C 180,E1 -4397.991,E2 -4397.991} C_VEL
LIN {X 0,Y 531.467,Z 351.076,A -85,B 0,C 180,E1 -4398.753,E2 -4398.753} C_VEL
LIN {X 0,Y 531.195,Z 361.545,A -85,B 0,C 180,E1 -4399.616,E2 -4399.616} C_VEL
LIN {X 0,Y 530.985,Z 370.108,A -85,B 0,C 180,E1 -4400.478,E2 -4400.478} C_VEL
LIN {X 0,Y 530.818,Z 378.012,A -85,B 0,C 180,E1 -4401.435,E2 -4401.435} C_VEL
LIN {X 0,Y 530.665,Z 385.734,A -85,B 0,C 180,E1 -4402.582,E2 -4402.582} C_VEL
LIN {X 0,Y 530.56,Z 392.853,A -85,B 0,C 180,E1 -4403.918,E2 -4403.918} C_VEL
LIN {X 0,Y 530.459,Z 397.589,A -85,B 0,C 180,E1 -4405.06,E2 -4405.06} C_VEL
LIN {X 0,Y 530.516,Z 401.212,A -85,B 0,C 180,E1 -4406.203,E2 -4406.203} C_VEL
LIN {X 0,Y 530.482,Z 403.078,A -85,B 0,C 180,E1 -4406.963,E2 -4406.963} C_VEL
LIN {X 0,Y 530.412,Z 404.475,A -85,B 0,C 180,E1 -4407.723,E2 -4407.723} C_VEL
LIN {X 0,Y 530.356,Z 406.081,A -85,B 0,C 180,E1 -4409.241,E2 -4409.241} C_VEL
LIN {X 0,Y 530.357,Z 406.297,A -85,B 0,C 180,E1 -4410.001,E2 -4410.001} C_VEL
LIN {X 0,Y 530.356,Z 406.08,A -85,B 0,C 180,E1 -4410.76,E2 -4410.76} C_VEL
LIN {X 0,Y 530.412,Z 404.473,A -85,B 0,C 180,E1 -4412.279,E2 -4412.279} C_VEL
LIN {X 0,Y 530.483,Z 403.075,A -85,B 0,C 180,E1 -4413.038,E2 -4413.038} C_VEL
LIN {X 0,Y 530.521,Z 400.129,A -85,B 0,C 180,E1 -4414.179,E2 -4414.179} C_VEL
LIN {X 0,Y 530.522,Z 396.139,A -85,B 0,C 180,E1 -4415.321,E2 -4415.321} C_VEL
LIN {X 0,Y 530.544,Z 390.674,A -85,B 0,C 180,E1 -4416.531,E2 -4416.531} C_VEL
LIN {X 0,Y 530.682,Z 384.548,A -85,B 0,C 180,E1 -4417.611,E2 -4417.611} C_VEL
LIN {X 0,Y 530.833,Z 376.492,A -85,B 0,C 180,E1 -4418.758,E2 -4418.758} C_VEL
LIN {X 0,Y 531.026,Z 368.287,A -85,B 0,C 180,E1 -4419.715,E2 -4419.715} C_VEL
LIN {X 0,Y 531.305,Z 358.285,A -85,B 0,C 180,E1 -4420.673,E2 -4420.673} C_VEL
LIN {X 0,Y 531.53,Z 346.851,A -85,B 0,C 180,E1 -4421.546,E2 -4421.546} C_VEL
LIN {X 0,Y 531.789,Z 335.935,A -85,B 0,C 180,E1 -4422.208,E2 -4422.208} C_VEL
LIN {X 0,Y 532.028,Z 323.685,A -85,B 0,C 180,E1 -4422.784,E2 -4422.784} C_VEL
LIN {X 0,Y 532.236,Z 310.833,A -85,B 0,C 180,E1 -4423.216,E2 -4423.216} C_VEL
LIN {X 0,Y 532.463,Z 297.21,A -85,B 0,C 180,E1 -4423.501,E2 -4423.501} C_VEL
LIN {X 0,Y 532.626,Z 202.5,A -85,B 0,C 180,E1 -4424.79,E2 -4424.79} C_VEL
LIN {X 0,Y 531.249,Z 192.979,A -85,B 0,C 180,E1 -4424.969,E2 -4424.969} C_VEL
LIN {X 0,Y 531.597,Z 173.239,A -85,B 0,C 180,E1 -4427.846,E2 -4427.846} C_VEL
LIN {X 0,Y 532.086,Z 149.862,A -85,B 0,C 180,E1 -4431.299,E2 -4431.299} C_VEL
LIN {X 0,Y 532.34,Z 134.967,A -85,B 0,C 180,E1 -4433.539,E2 -4433.539} C_VEL
LIN {X 0,Y 531.041,Z 127.336,A -85,B 0,C 180,E1 -4434.795,E2 -4434.795} C_VEL
LIN {X 0,Y 530.976,Z 127.345,A -85,B 0,C 180,E1 -4437.598,E2 -4437.598} C_VEL
LIN {X 0,Y 530.962,Z 127.35,A -85,B 0,C 180,E1 -4440.198,E2 -4440.198} C_VEL
LIN {X 0,Y 530.97,Z 127.342,A -85,B 0,C 180,E1 -4442.867,E2 -4442.867} C_VEL
LIN {X 0,Y 530.953,Z 127.349,A -85,B 0,C 180,E1 -4445.62,E2 -4445.62} C_VEL
LIN {X 0,Y 530.967,Z 127.34,A -85,B 0,C 180,E1 -4448.653,E2 -4448.653} C_VEL
LIN {X 0,Y 530.988,Z 127.345,A -85,B 0,C 180,E1 -4451.436,E2 -4451.436} C_VEL
LIN {X 0,Y 530.972,Z 127.34,A -85,B 0,C 180,E1 -4454.549,E2 -4454.549} C_VEL
LIN {X 0,Y 530.968,Z 127.344,A -85,B 0,C 180,E1 -4457.836,E2 -4457.836} C_VEL
LIN {X 0,Y 530.97,Z 127.342,A -85,B 0,C 180,E1 -4460.555,E2 -4460.555} C_VEL
LIN {X 0,Y 530.953,Z 127.348,A -85,B 0,C 180,E1 -4463.441,E2 -4463.441} C_VEL
LIN {X 0,Y 530.962,Z 127.344,A -85,B 0,C 180,E1 -4466.5,E2 -4466.5} C_VEL
LIN {X 0,Y 530.955,Z 127.346,A -85,B 0,C 180,E1 -4469.359,E2 -4469.359} C_VEL
LIN {X 0,Y 530.959,Z 127.344,A -85,B 0,C 180,E1 -4472.401,E2 -4472.401} C_VEL
LIN {X 0,Y 530.948,Z 127.35,A -85,B 0,C 180,E1 -4474.939,E2 -4474.939} C_VEL
LIN {X 0,Y 530.971,Z 127.341,A -85,B 0,C 180,E1 -4477.9,E2 -4477.9} C_VEL
LIN {X 0,Y 530.96,Z 127.347,A -85,B 0,C 180,E1 -4480.676,E2 -4480.676} C_VEL
LIN {X 0,Y 530.935,Z 127.346,A -85,B 0,C 180,E1 -4483.069,E2 -4483.069} C_VEL
LIN {X 0,Y 530.996,Z 127.335,A -85,B 0,C 180,E1 -4485.435,E2 -4485.435} C_VEL
LIN {X 0,Y 530.983,Z 127.344,A -85,B 0,C 180,E1 -4488.549,E2 -4488.549} C_VEL
LIN {X 0,Y 530.976,Z 127.338,A -85,B 0,C 180,E1 -4491.628,E2 -4491.628} C_VEL
LIN {X 0,Y 531.077,Z 127.328,A -85,B 0,C 180,E1 -4494.685,E2 -4494.685} C_VEL
LIN {X 0,Y 531.13,Z 127.322,A -85,B 0,C 180,E1 -4497.725,E2 -4497.725} C_VEL
LIN {X 0,Y 531.126,Z 127.328,A -85,B 0,C 180,E1 -4500,E2 -4500} C_VEL
LIN {X 0,Y 531.131,Z 127.32,A -85,B 0,C 180,E1 -4502.275,E2 -4502.275} C_VEL
LIN {X 0,Y 531.082,Z 127.329,A -85,B 0,C 180,E1 -4505.315,E2 -4505.315} C_VEL
LIN {X 0,Y 531.028,Z 127.33,A -85,B 0,C 180,E1 -4508.371,E2 -4508.371} C_VEL
LIN {X 0,Y 531.048,Z 127.337,A -85,B 0,C 180,E1 -4511.67,E2 -4511.67} C_VEL
LIN {X 0,Y 531.019,Z 127.334,A -85,B 0,C 180,E1 -4514.951,E2 -4514.951} C_VEL
LIN {X 0,Y 530.979,Z 127.341,A -85,B 0,C 180,E1 -4517.724,E2 -4517.724} C_VEL
LIN {X 0,Y 531.025,Z 127.332,A -85,B 0,C 180,E1 -4520.127,E2 -4520.127} C_VEL
LIN {X 0,Y 530.941,Z 127.346,A -85,B 0,C 180,E1 -4522.574,E2 -4522.574} C_VEL
LIN {X 0,Y 530.954,Z 127.349,A -85,B 0,C 180,E1 -4525.06,E2 -4525.06} C_VEL
LIN {X 0,Y 530.973,Z 127.34,A -85,B 0,C 180,E1 -4527.598,E2 -4527.598} C_VEL
LIN {X 0,Y 530.954,Z 127.343,A -85,B 0,C 180,E1 -4530.198,E2 -4530.198} C_VEL
LIN {X 0,Y 530.967,Z 127.348,A -85,B 0,C 180,E1 -4532.867,E2 -4532.867} C_VEL
LIN {X 0,Y 530.955,Z 127.342,A -85,B 0,C 180,E1 -4535.62,E2 -4535.62} C_VEL
LIN {X 0,Y 530.966,Z 127.347,A -85,B 0,C 180,E1 -4538.653,E2 -4538.653} C_VEL
LIN {X 0,Y 530.995,Z 127.333,A -85,B 0,C 180,E1 -4541.436,E2 -4541.436} C_VEL
LIN {X 0,Y 530.956,Z 127.342,A -85,B 0,C 180,E1 -4543.522,E2 -4543.522} C_VEL
LIN {X 0,Y 530.279,Z 127.433,A -85,B 0,C 180,E1 -4544.156,E2 -4544.156} C_VEL
LIN {X 0,Y 527.426,Z 127.787,A -85,B 0,C 180,E1 -4545.184,E2 -4545.184} C_VEL
LIN {X 0,Y 525.021,Z 128.087,A -85,B 0,C 180,E1 -4546.013,E2 -4546.013} C_VEL
LIN {X 0,Y 523.988,Z 128.215,A -85,B 0,C 180,E1 -4546.652,E2 -4546.652} C_VEL
LIN {X 0,Y 523.904,Z 128.222,A -85,B 0,C 180,E1 -4546.869,E2 -4546.869} C_VEL
LIN {X 0,Y 523.94,Z 128.217,A -85,B 0,C 180,E1 -4548.908,E2 -4548.908} C_VEL
LIN {X 0,Y 523.919,Z 128.225,A -85,B 0,C 180,E1 -4551.898,E2 -4551.898} C_VEL
LIN {X 0,Y 523.928,Z 128.218,A -85,B 0,C 180,E1 -4554.911,E2 -4554.911} C_VEL
LIN {X 0,Y 523.939,Z 128.222,A -85,B 0,C 180,E1 -4557.68,E2 -4557.68} C_VEL
LIN {X 0,Y 523.958,Z 128.216,A -85,B 0,C 180,E1 -4560.677,E2 -4560.677} C_VEL
LIN {X 0,Y 523.977,Z 128.221,A -85,B 0,C 180,E1 -4563.728,E2 -4563.728} C_VEL
LIN {X 0,Y 524.008,Z 128.392,A -85,B 0,C 180,E1 -4566.059,E2 -4566.059} C_VEL
LIN {X 0,Y 524.447,Z 132.714,A -85,B 0,C 180,E1 -4566.922,E2 -4566.922} C_VEL
LIN {X 0,Y 524.258,Z 148.138,A -85,B 0,C 180,E1 -4569.899,E2 -4569.899} C_VEL
LIN {X 0,Y 525.985,Z 158.424,A -85,B 0,C 180,E1 -4570.1,E2 -4570.1} C_VEL
LIN {X 0,Y 525.547,Z 255.08,A -85,B 0,C 180,E1 -4571.445,E2 -4571.445} C_VEL
LIN {X 0,Y 525.347,Z 268.361,A -85,B 0,C 180,E1 -4571.79,E2 -4571.79} C_VEL
LIN {X 0,Y 525.165,Z 280.89,A -85,B 0,C 180,E1 -4572.274,E2 -4572.274} C_VEL
LIN {X 0,Y 524.944,Z 292.272,A -85,B 0,C 180,E1 -4572.87,E2 -4572.87} C_VEL
LIN {X 0,Y 524.653,Z 303.99,A -85,B 0,C 180,E1 -4573.661,E2 -4573.661} C_VEL
LIN {X 0,Y 524.359,Z 314.469,A -85,B 0,C 180,E1 -4574.549,E2 -4574.549} C_VEL
LIN {X 0,Y 524.164,Z 323.029,A -85,B 0,C 180,E1 -4575.439,E2 -4575.439} C_VEL
LIN {X 0,Y 523.87,Z 332.223,A -85,B 0,C 180,E1 -4576.619,E2 -4576.619} C_VEL
LIN {X 0,Y 523.714,Z 339.592,A -85,B 0,C 180,E1 -4577.798,E2 -4577.798} C_VEL
LIN {X 0,Y 523.582,Z 344.71,A -85,B 0,C 180,E1 -4578.808,E2 -4578.808} C_VEL
LIN {X 0,Y 523.496,Z 349.365,A -85,B 0,C 180,E1 -4579.948,E2 -4579.948} C_VEL
LIN {X 0,Y 523.404,Z 353.035,A -85,B 0,C 180,E1 -4581.116,E2 -4581.116} C_VEL
LIN {X 0,Y 523.384,Z 355.677,A -85,B 0,C 180,E1 -4582.282,E2 -4582.282} C_VEL
LIN {X 0,Y 523.441,Z 357.419,A -85,B 0,C 180,E1 -4583.499,E2 -4583.499} C_VEL
LIN {X 0,Y 523.379,Z 358.152,A -85,B 0,C 180,E1 -4584.606,E2 -4584.606} C_VEL
LIN {X 0,Y 523.402,Z 357.812,A -85,B 0,C 180,E1 -4586.15,E2 -4586.15} C_VEL
LIN {X 0,Y 523.439,Z 357.063,A -85,B 0,C 180,E1 -4586.921,E2 -4586.921} C_VEL
LIN {X 0,Y 523.301,Z 354.312,A -85,B 0,C 180,E1 -4588.46,E2 -4588.46} C_VEL
LIN {X 0,Y 523.416,Z 351.142,A -85,B 0,C 180,E1 -4589.615,E2 -4589.615} C_VEL
LIN {X 0,Y 523.431,Z 346.939,A -85,B 0,C 180,E1 -4590.769,E2 -4590.769} C_VEL
LIN {X 0,Y 523.643,Z 341.563,A -85,B 0,C 180,E1 -4591.922,E2 -4591.922} C_VEL
LIN {X 0,Y 523.693,Z 334.878,A -85,B 0,C 180,E1 -4593.076,E2 -4593.076} C_VEL
LIN {X 0,Y 524.019,Z 326.542,A -85,B 0,C 180,E1 -4594.229,E2 -4594.229} C_VEL
LIN {X 0,Y 524.239,Z 317.992,A -85,B 0,C 180,E1 -4595.191,E2 -4595.191} C_VEL
LIN {X 0,Y 524.551,Z 307.475,A -85,B 0,C 180,E1 -4596.152,E2 -4596.152} C_VEL
LIN {X 0,Y 524.859,Z 297.026,A -85,B 0,C 180,E1 -4596.921,E2 -4596.921} C_VEL
LIN {X 0,Y 525.12,Z 285.856,A -85,B 0,C 180,E1 -4597.572,E2 -4597.572} C_VEL
LIN {X 0,Y 525.292,Z 273.398,A -85,B 0,C 180,E1 -4598.123,E2 -4598.123} C_VEL
LIN {X 0,Y 525.496,Z 260.226,A -85,B 0,C 180,E1 -4598.532,E2 -4598.532} C_VEL
LIN {X 0,Y 525.556,Z 247.246,A -85,B 0,C 180,E1 -4598.773,E2 -4598.773} C_VEL
LIN {X 0,Y 525.915,Z 156.968,A -85,B 0,C 180,E1 -4600.012,E2 -4600.012} C_VEL
LIN {X 0,Y 524.203,Z 148.05,A -85,B 0,C 180,E1 -4600.207,E2 -4600.207} C_VEL
LIN {X 0,Y 524.419,Z 132.747,A -85,B 0,C 180,E1 -4603.168,E2 -4603.168} C_VEL
LIN {X 0,Y 523.979,Z 128.219,A -85,B 0,C 180,E1 -4604.119,E2 -4604.119} C_VEL
LIN {X 0,Y 523.956,Z 128.216,A -85,B 0,C 180,E1 -4607.162,E2 -4607.162} C_VEL
LIN {X 0,Y 523.973,Z 128.219,A -85,B 0,C 180,E1 -4610.409,E2 -4610.409} C_VEL
LIN {X 0,Y 523.911,Z 128.221,A -85,B 0,C 180,E1 -4612.892,E2 -4612.892} C_VEL
LIN {X 0,Y 523.983,Z 128.218,A -85,B 0,C 180,E1 -4616.018,E2 -4616.018} C_VEL
LIN {X 0,Y 523.927,Z 128.218,A -85,B 0,C 180,E1 -4618.874,E2 -4618.874} C_VEL
LIN {X 0,Y 523.919,Z 128.223,A -85,B 0,C 180,E1 -4621.543,E2 -4621.543} C_VEL
LIN {X 0,Y 523.929,Z 128.221,A -85,B 0,C 180,E1 -4624.289,E2 -4624.289} C_VEL
LIN {X 0,Y 523.903,Z 128.223,A -85,B 0,C 180,E1 -4627.131,E2 -4627.131} C_VEL
LIN {X 0,Y 523.933,Z 128.22,A -85,B 0,C 180,E1 -4630.129,E2 -4630.129} C_VEL
LIN {X 0,Y 523.929,Z 128.219,A -85,B 0,C 180,E1 -4632.458,E2 -4632.458} C_VEL
LIN {X 0,Y 523.937,Z 128.223,A -85,B 0,C 180,E1 -4635.309,E2 -4635.309} C_VEL
LIN {X 0,Y 523.948,Z 128.218,A -85,B 0,C 180,E1 -4638.689,E2 -4638.689} C_VEL
LIN {X 0,Y 523.908,Z 128.226,A -85,B 0,C 180,E1 -4641.08,E2 -4641.08} C_VEL
LIN {X 0,Y 523.891,Z 128.225,A -85,B 0,C 180,E1 -4643.824,E2 -4643.824} C_VEL
LIN {X 0,Y 523.904,Z 128.225,A -85,B 0,C 180,E1 -4646.633,E2 -4646.633} C_VEL
LIN {X 0,Y 523.938,Z 128.222,A -85,B 0,C 180,E1 -4649.354,E2 -4649.354} C_VEL
LIN {X 0,Y 523.962,Z 128.216,A -85,B 0,C 180,E1 -4652.282,E2 -4652.282} C_VEL
LIN {X 0,Y 523.891,Z 128.225,A -85,B 0,C 180,E1 -4655.426,E2 -4655.426} C_VEL
LIN {X 0,Y 523.925,Z 128.22,A -85,B 0,C 180,E1 -4657.939,E2 -4657.939} C_VEL
LIN {X 0,Y 523.955,Z 128.221,A -85,B 0,C 180,E1 -4660.407,E2 -4660.407} C_VEL
LIN {X 0,Y 523.917,Z 128.225,A -85,B 0,C 180,E1 -4662.835,E2 -4662.835} C_VEL
LIN {X 0,Y 523.95,Z 128.217,A -85,B 0,C 180,E1 -4665.235,E2 -4665.235} C_VEL
LIN {X 0,Y 524.001,Z 128.215,A -85,B 0,C 180,E1 -4668.394,E2 -4668.394} C_VEL
LIN {X 0,Y 523.97,Z 128.215,A -85,B 0,C 180,E1 -4671.515,E2 -4671.515} C_VEL
LIN {X 0,Y 524.021,Z 128.211,A -85,B 0,C 180,E1 -4674.613,E2 -4674.613} C_VEL
LIN {X 0,Y 524.092,Z 128.203,A -85,B 0,C 180,E1 -4677.694,E2 -4677.694} C_VEL
LIN {X 0,Y 524.084,Z 128.205,A -85,B 0,C 180,E1 -4680,E2 -4680} C_VEL
LIN {X 0,Y 524.092,Z 128.202,A -85,B 0,C 180,E1 -4682.306,E2 -4682.306} C_VEL
LIN {X 0,Y 524.008,Z 128.213,A -85,B 0,C 180,E1 -4686.159,E2 -4686.159} C_VEL
LIN {X 0,Y 523.967,Z 128.218,A -85,B 0,C 180,E1 -4689.262,E2 -4689.262} C_VEL
LIN {X 0,Y 523.985,Z 128.217,A -85,B 0,C 180,E1 -4691.737,E2 -4691.737} C_VEL
LIN {X 0,Y 523.971,Z 128.217,A -85,B 0,C 180,E1 -4695.048,E2 -4695.048} C_VEL
LIN {X 0,Y 523.931,Z 128.22,A -85,B 0,C 180,E1 -4697.97,E2 -4697.97} C_VEL
LIN {X 0,Y 523.945,Z 128.217,A -85,B 0,C 180,E1 -4700.411,E2 -4700.411} C_VEL
LIN {X 0,Y 523.895,Z 128.227,A -85,B 0,C 180,E1 -4702.894,E2 -4702.894} C_VEL
LIN {X 0,Y 523.895,Z 128.227,A -85,B 0,C 180,E1 -4705.422,E2 -4705.422} C_VEL
LIN {X 0,Y 523.946,Z 128.217,A -85,B 0,C 180,E1 -4708,E2 -4708} C_VEL
LIN {X 0,Y 523.929,Z 128.226,A -85,B 0,C 180,E1 -4710.854,E2 -4710.854} C_VEL
LIN {X 0,Y 523.92,Z 128.22,A -85,B 0,C 180,E1 -4713.73,E2 -4713.73} C_VEL
LIN {X 0,Y 523.894,Z 128.226,A -85,B 0,C 180,E1 -4716.402,E2 -4716.402} C_VEL
LIN {X 0,Y 523.911,Z 128.224,A -85,B 0,C 180,E1 -4719.086,E2 -4719.086} C_VEL
LIN {X 0,Y 523.943,Z 128.219,A -85,B 0,C 180,E1 -4722.12,E2 -4722.12} C_VEL
LIN {X 0,Y 523.936,Z 128.218,A -85,B 0,C 180,E1 -4725.311,E2 -4725.311} C_VEL
LIN {X 0,Y 523.949,Z 128.22,A -85,B 0,C 180,E1 -4728.691,E2 -4728.691} C_VEL
LIN {X 0,Y 523.913,Z 128.22,A -85,B 0,C 180,E1 -4731.081,E2 -4731.081} C_VEL
LIN {X 0,Y 523.895,Z 128.225,A -85,B 0,C 180,E1 -4733.826,E2 -4733.826} C_VEL
LIN {X 0,Y 523.937,Z 128.219,A -85,B 0,C 180,E1 -4736.637,E2 -4736.637} C_VEL
LIN {X 0,Y 523.953,Z 128.215,A -85,B 0,C 180,E1 -4739.357,E2 -4739.357} C_VEL
LIN {X 0,Y 523.976,Z 128.217,A -85,B 0,C 180,E1 -4742.282,E2 -4742.282} C_VEL
LIN {X 0,Y 523.994,Z 128.268,A -85,B 0,C 180,E1 -4745.089,E2 -4745.089} C_VEL
LIN {X 0,Y 525.384,Z 136.026,A -85,B 0,C 180,E1 -4746.341,E2 -4746.341} C_VEL
LIN {X 0,Y 525.118,Z 150.974,A -85,B 0,C 180,E1 -4748.612,E2 -4748.612} C_VEL
LIN {X 0,Y 524.6,Z 173.957,A -85,B 0,C 180,E1 -4752.055,E2 -4752.055} C_VEL
LIN {X 0,Y 524.233,Z 192.668,A -85,B 0,C 180,E1 -4754.824,E2 -4754.824} C_VEL
LIN {X 0,Y 525.879,Z 204.768,A -85,B 0,C 180,E1 -4755.052,E2 -4755.052} C_VEL
LIN {X 0,Y 525.488,Z 301.345,A -85,B 0,C 180,E1 -4756.391,E2 -4756.391} C_VEL
LIN {X 0,Y 525.294,Z 313.876,A -85,B 0,C 180,E1 -4756.707,E2 -4756.707} C_VEL
LIN {X 0,Y 525.007,Z 326.824,A -85,B 0,C 180,E1 -4757.191,E2 -4757.191} C_VEL
LIN {X 0,Y 524.737,Z 339.264,A -85,B 0,C 180,E1 -4757.832,E2 -4757.832} C_VEL
LIN {X 0,Y 524.478,Z 350.751,A -85,B 0,C 180,E1 -4758.601,E2 -4758.601} C_VEL
LIN {X 0,Y 524.2,Z 361.221,A -85,B 0,C 180,E1 -4759.475,E2 -4759.475} C_VEL
LIN {X 0,Y 523.947,Z 369.784,A -85,B 0,C 180,E1 -4760.349,E2 -4760.349} C_VEL
LIN {X 0,Y 523.738,Z 377.687,A -85,B 0,C 180,E1 -4761.318,E2 -4761.318} C_VEL
LIN {X 0,Y 523.576,Z 385.409,A -85,B 0,C 180,E1 -4762.481,E2 -4762.481} C_VEL
LIN {X 0,Y 523.458,Z 392.529,A -85,B 0,C 180,E1 -4763.835,E2 -4763.835} C_VEL
LIN {X 0,Y 523.383,Z 397.266,A -85,B 0,C 180,E1 -4764.994,E2 -4764.994} C_VEL
LIN {X 0,Y 523.443,Z 400.89,A -85,B 0,C 180,E1 -4766.151,E2 -4766.151} C_VEL
LIN {X 0,Y 523.39,Z 402.755,A -85,B 0,C 180,E1 -4766.922,E2 -4766.922} C_VEL
LIN {X 0,Y 523.337,Z 404.153,A -85,B 0,C 180,E1 -4767.692,E2 -4767.692} C_VEL
LIN {X 0,Y 523.263,Z 405.758,A -85,B 0,C 180,E1 -4769.231,E2 -4769.231} C_VEL
LIN {X 0,Y 523.265,Z 405.974,A -85,B 0,C 180,E1 -4770.001,E2 -4770.001} C_VEL
LIN {X 0,Y 523.275,Z 405.146,A -85,B 0,C 180,E1 -4771.54,E2 -4771.54} C_VEL
LIN {X 0,Y 523.337,Z 404.149,A -85,B 0,C 180,E1 -4772.31,E2 -4772.31} C_VEL
LIN {X 0,Y 523.391,Z 402.749,A -85,B 0,C 180,E1 -4773.08,E2 -4773.08} C_VEL
LIN {X 0,Y 523.422,Z 399.803,A -85,B 0,C 180,E1 -4774.236,E2 -4774.236} C_VEL
LIN {X 0,Y 523.456,Z 395.813,A -85,B 0,C 180,E1 -4775.393,E2 -4775.393} C_VEL
LIN {X 0,Y 523.502,Z 389.759,A -85,B 0,C 180,E1 -4776.731,E2 -4776.731} C_VEL
LIN {X 0,Y 523.644,Z 382.978,A -85,B 0,C 180,E1 -4777.908,E2 -4777.908} C_VEL
LIN {X 0,Y 523.82,Z 374.666,A -85,B 0,C 180,E1 -4779.071,E2 -4779.071} C_VEL
LIN {X 0,Y 524.016,Z 366.149,A -85,B 0,C 180,E1 -4780.042,E2 -4780.042} C_VEL
